LIN {X 0,Y 339.531,Z 433.374,A -85,B 0,C 180,E1 -14042.372,E2 -14042.372} C_VEL
LIN {X 0,Y 339.69,Z 432.812,A -85,B 0,C 180,E1 -14044.747,E2 -14044.747} C_VEL
LIN {X 0,Y 340.181,Z 431.007,A -85,B 0,C 180,E1 -14047.12,E2 -14047.12} C_VEL
LIN {X 0,Y 340.922,Z 427.934,A -85,B 0,C 180,E1 -14049.492,E2 -14049.492} C_VEL
LIN {X 0,Y 341.879,Z 423.539,A -85,B 0,C 180,E1 -14051.863,E2 -14051.863} C_VEL
LIN {X 0,Y 343.294,Z 417.733,A -85,B 0,C 180,E1 -14054.221,E2 -14054.221} C_VEL
LIN {X 0,Y 344.568,Z 412.354,A -85,B 0,C 180,E1 -14055.983,E2 -14055.983} C_VEL
LIN {X 0,Y 346.771,Z 403.681,A -85,B 0,C 180,E1 -14058.308,E2 -14058.308} C_VEL
LIN {X 0,Y 348.941,Z 394.494,A -85,B 0,C 180,E1 -14060.33,E2 -14060.33} C_VEL
LIN {X 0,Y 351.488,Z 383.498,A -85,B 0,C 180,E1 -14062.327,E2 -14062.327} C_VEL
LIN {X 0,Y 354.287,Z 371.267,A -85,B 0,C 180,E1 -14064.146,E2 -14064.146} C_VEL
LIN {X 0,Y 356.805,Z 358.929,A -85,B 0,C 180,E1 -14065.679,E2 -14065.679} C_VEL
LIN {X 0,Y 359.387,Z 345.597,A -85,B 0,C 180,E1 -14067.043,E2 -14067.043} C_VEL
LIN {X 0,Y 361.83,Z 331.122,A -85,B 0,C 180,E1 -14068.258,E2 -14068.258} C_VEL
LIN {X 0,Y 364.103,Z 316.147,A -85,B 0,C 180,E1 -14069.253,E2 -14069.253} C_VEL
LIN {X 0,Y 366.036,Z 300.525,A -85,B 0,C 180,E1 -14070.067,E2 -14070.067} C_VEL
LIN {X 0,Y 367.961,Z 282.022,A -85,B 0,C 180,E1 -14070.767,E2 -14070.767} C_VEL
LIN {X 0,Y 375.63,Z 216.607,A -85,B 0,C 180,E1 -14073.03,E2 -14073.03} C_VEL
LIN {X 0,Y 379.653,Z 185.862,A -85,B 0,C 180,E1 -14074.119,E2 -14074.119} C_VEL
LIN {X 0,Y 376.328,Z 179.523,A -85,B 0,C 180,E1 -14075.526,E2 -14075.526} C_VEL
LIN {X 0,Y 373.796,Z 175.547,A -85,B 0,C 180,E1 -14076.722,E2 -14076.722} C_VEL
LIN {X 0,Y 371.547,Z 172.279,A -85,B 0,C 180,E1 -14077.969,E2 -14077.969} C_VEL
LIN {X 0,Y 369.521,Z 169.583,A -85,B 0,C 180,E1 -14079.332,E2 -14079.332} C_VEL
LIN {X 0,Y 367.108,Z 166.762,A -85,B 0,C 180,E1 -14081.701,E2 -14081.701} C_VEL
LIN {X 0,Y 365.993,Z 166.623,A -85,B 0,C 180,E1 -14083.732,E2 -14083.732} C_VEL
LIN {X 0,Y 365.943,Z 167.567,A -85,B 0,C 180,E1 -14085.646,E2 -14085.646} C_VEL
LIN {X 0,Y 366.76,Z 169.742,A -85,B 0,C 180,E1 -14087.516,E2 -14087.516} C_VEL
LIN {X 0,Y 368.364,Z 172.942,A -85,B 0,C 180,E1 -14089.299,E2 -14089.299} C_VEL
LIN {X 0,Y 371.418,Z 179.732,A -85,B 0,C 180,E1 -14091.59,E2 -14091.59} C_VEL
LIN {X 0,Y 374.03,Z 186.01,A -85,B 0,C 180,E1 -14093.104,E2 -14093.104} C_VEL
LIN {X 0,Y 376.608,Z 193.132,A -85,B 0,C 180,E1 -14094.421,E2 -14094.421} C_VEL
LIN {X 0,Y 377.224,Z 207.224,A -85,B 0,C 180,E1 -14095.553,E2 -14095.553} C_VEL
LIN {X 0,Y 377.182,Z 212.766,A -85,B 0,C 180,E1 -14095.905,E2 -14095.905} C_VEL
LIN {X 0,Y 368.41,Z 287.792,A -85,B 0,C 180,E1 -14098.479,E2 -14098.479} C_VEL
LIN {X 0,Y 364.577,Z 324.529,A -85,B 0,C 180,E1 -14099.76,E2 -14099.76} C_VEL
LIN {X 0,Y 362.084,Z 341.748,A -85,B 0,C 180,E1 -14100.573,E2 -14100.573} C_VEL
LIN {X 0,Y 359.351,Z 357.417,A -85,B 0,C 180,E1 -14101.529,E2 -14101.529} C_VEL
LIN {X 0,Y 356.653,Z 371.828,A -85,B 0,C 180,E1 -14102.646,E2 -14102.646} C_VEL
LIN {X 0,Y 353.636,Z 386.742,A -85,B 0,C 180,E1 -14104.073,E2 -14104.073} C_VEL
LIN {X 0,Y 350.88,Z 399.866,A -85,B 0,C 180,E1 -14105.6,E2 -14105.6} C_VEL
LIN {X 0,Y 348.084,Z 412.984,A -85,B 0,C 180,E1 -14107.442,E2 -14107.442} C_VEL
LIN {X 0,Y 345.654,Z 424.786,A -85,B 0,C 180,E1 -14109.445,E2 -14109.445} C_VEL
LIN {X 0,Y 343.653,Z 435.782,A -85,B 0,C 180,E1 -14111.519,E2 -14111.519} C_VEL
LIN {X 0,Y 342.125,Z 444.941,A -85,B 0,C 180,E1 -14113.593,E2 -14113.593} C_VEL
LIN {X 0,Y 340.95,Z 452.532,A -85,B 0,C 180,E1 -14115.679,E2 -14115.679} C_VEL
LIN {X 0,Y 340.039,Z 459.612,A -85,B 0,C 180,E1 -14118.072,E2 -14118.072} C_VEL
LIN {X 0,Y 339.417,Z 465.159,A -85,B 0,C 180,E1 -14120.465,E2 -14120.465} C_VEL
LIN {X 0,Y 339.169,Z 469.321,A -85,B 0,C 180,E1 -14122.858,E2 -14122.858} C_VEL
LIN {X 0,Y 339.05,Z 472.204,A -85,B 0,C 180,E1 -14125.244,E2 -14125.244} C_VEL
LIN {X 0,Y 339.04,Z 473.874,A -85,B 0,C 180,E1 -14127.624,E2 -14127.624} C_VEL
LIN {X 0,Y 339.07,Z 474.355,A -85,B 0,C 180,E1 -14130,E2 -14130} C_VEL
LIN {X 0,Y 339.041,Z 473.645,A -85,B 0,C 180,E1 -14132.376,E2 -14132.376} C_VEL
LIN {X 0,Y 339.064,Z 471.711,A -85,B 0,C 180,E1 -14134.756,E2 -14134.756} C_VEL
LIN {X 0,Y 339.22,Z 468.501,A -85,B 0,C 180,E1 -14137.141,E2 -14137.141} C_VEL
LIN {X 0,Y 339.362,Z 463.965,A -85,B 0,C 180,E1 -14139.537,E2 -14139.537} C_VEL
LIN {X 0,Y 339.951,Z 458.003,A -85,B 0,C 180,E1 -14141.931,E2 -14141.931} C_VEL
LIN {X 0,Y 340.726,Z 450.427,A -85,B 0,C 180,E1 -14144.331,E2 -14144.331} C_VEL
LIN {X 0,Y 341.897,Z 442.263,A -85,B 0,C 180,E1 -14146.418,E2 -14146.418} C_VEL
LIN {X 0,Y 344.5,Z 427.37,A -85,B 0,C 180,E1 -14149.67,E2 -14149.67} C_VEL
LIN {X 0,Y 346.677,Z 416.152,A -85,B 0,C 180,E1 -14151.714,E2 -14151.714} C_VEL
LIN {X 0,Y 349.347,Z 403.732,A -85,B 0,C 180,E1 -14153.568,E2 -14153.568} C_VEL
LIN {X 0,Y 352.146,Z 390.155,A -85,B 0,C 180,E1 -14155.252,E2 -14155.252} C_VEL
LIN {X 0,Y 355.058,Z 375.843,A -85,B 0,C 180,E1 -14156.695,E2 -14156.695} C_VEL
LIN {X 0,Y 357.887,Z 360.455,A -85,B 0,C 180,E1 -14157.972,E2 -14157.972} C_VEL
LIN {X 0,Y 360.631,Z 344.612,A -85,B 0,C 180,E1 -14158.997,E2 -14158.997} C_VEL
LIN {X 0,Y 363.283,Z 326.693,A -85,B 0,C 180,E1 -14159.878,E2 -14159.878} C_VEL
LIN {X 0,Y 365.647,Z 304.905,A -85,B 0,C 180,E1 -14160.66,E2 -14160.66} C_VEL
LIN {X 0,Y 373.572,Z 232.695,A -85,B 0,C 180,E1 -14163.138,E2 -14163.138} C_VEL
LIN {X 0,Y 376.754,Z 206.525,A -85,B 0,C 180,E1 -14164.063,E2 -14164.063} C_VEL
LIN {X 0,Y 377.117,Z 189.528,A -85,B 0,C 180,E1 -14165.126,E2 -14165.126} C_VEL
LIN {X 0,Y 377.037,Z 185.508,A -85,B 0,C 180,E1 -14165.437,E2 -14165.437} C_VEL
LIN {X 0,Y 374.782,Z 174.187,A -85,B 0,C 180,E1 -14167.011,E2 -14167.011} C_VEL
LIN {X 0,Y 372.206,Z 169.945,A -85,B 0,C 180,E1 -14168.343,E2 -14168.343} C_VEL
LIN {X 0,Y 370.361,Z 166.78,A -85,B 0,C 180,E1 -14169.51,E2 -14169.51} C_VEL
LIN {X 0,Y 367.673,Z 162.482,A -85,B 0,C 180,E1 -14171.8,E2 -14171.8} C_VEL
LIN {X 0,Y 366.032,Z 160.666,A -85,B 0,C 180,E1 -14174.345,E2 -14174.345} C_VEL
LIN {X 0,Y 365.952,Z 160.508,A -85,B 0,C 180,E1 -14176.262,E2 -14176.262} C_VEL
LIN {X 0,Y 366.717,Z 161.339,A -85,B 0,C 180,E1 -14178.083,E2 -14178.083} C_VEL
LIN {X 0,Y 368.403,Z 163.16,A -85,B 0,C 180,E1 -14179.91,E2 -14179.91} C_VEL
LIN {X 0,Y 370.56,Z 166.521,A -85,B 0,C 180,E1 -14181.597,E2 -14181.597} C_VEL
LIN {X 0,Y 373.531,Z 171.452,A -85,B 0,C 180,E1 -14183.332,E2 -14183.332} C_VEL
LIN {X 0,Y 375.997,Z 175.941,A -85,B 0,C 180,E1 -14184.535,E2 -14184.535} C_VEL
LIN {X 0,Y 379.423,Z 182.777,A -85,B 0,C 180,E1 -14185.992,E2 -14185.992} C_VEL
LIN {X 0,Y 369.991,Z 258.966,A -85,B 0,C 180,E1 -14188.629,E2 -14188.629} C_VEL
LIN {X 0,Y 366.125,Z 295.865,A -85,B 0,C 180,E1 -14189.909,E2 -14189.909} C_VEL
LIN {X 0,Y 364.358,Z 311.193,A -85,B 0,C 180,E1 -14190.642,E2 -14190.642} C_VEL
LIN {X 0,Y 362.129,Z 326.807,A -85,B 0,C 180,E1 -14191.61,E2 -14191.61} C_VEL
LIN {X 0,Y 359.897,Z 340.486,A -85,B 0,C 180,E1 -14192.684,E2 -14192.684} C_VEL
LIN {X 0,Y 357.363,Z 354.596,A -85,B 0,C 180,E1 -14194.051,E2 -14194.051} C_VEL
LIN {X 0,Y 354.988,Z 366.509,A -85,B 0,C 180,E1 -14195.433,E2 -14195.433} C_VEL
LIN {X 0,Y 352.176,Z 379.037,A -85,B 0,C 180,E1 -14197.171,E2 -14197.171} C_VEL
LIN {X 0,Y 349.605,Z 390.384,A -85,B 0,C 180,E1 -14199.095,E2 -14199.095} C_VEL
LIN {X 0,Y 347.647,Z 398.906,A -85,B 0,C 180,E1 -14200.822,E2 -14200.822} C_VEL
LIN {X 0,Y 345.627,Z 407.42,A -85,B 0,C 180,E1 -14202.882,E2 -14202.882} C_VEL
LIN {X 0,Y 344.03,Z 413.434,A -85,B 0,C 180,E1 -14204.6,E2 -14204.6} C_VEL
LIN {X 0,Y 342.6,Z 420.079,A -85,B 0,C 180,E1 -14206.959,E2 -14206.959} C_VEL
LIN {X 0,Y 341.42,Z 425.246,A -85,B 0,C 180,E1 -14209.324,E2 -14209.324} C_VEL
LIN {X 0,Y 340.504,Z 429.044,A -85,B 0,C 180,E1 -14211.693,E2 -14211.693} C_VEL
LIN {X 0,Y 339.786,Z 431.564,A -85,B 0,C 180,E1 -14214.064,E2 -14214.064} C_VEL
LIN {X 0,Y 339.631,Z 432.805,A -85,B 0,C 180,E1 -14216.441,E2 -14216.441} C_VEL
LIN {X 0,Y 339.363,Z 432.834,A -85,B 0,C 180,E1 -14218.814,E2 -14218.814} C_VEL
LIN {X 0,Y 339.27,Z 431.606,A -85,B 0,C 180,E1 -14221.187,E2 -14221.187} C_VEL
LIN {X 0,Y 339.294,Z 429.111,A -85,B 0,C 180,E1 -14223.563,E2 -14223.563} C_VEL
LIN {X 0,Y 339.449,Z 425.282,A -85,B 0,C 180,E1 -14225.942,E2 -14225.942} C_VEL
LIN {X 0,Y 339.686,Z 421.495,A -85,B 0,C 180,E1 -14227.729,E2 -14227.729} C_VEL
LIN {X 0,Y 340.078,Z 415.107,A -85,B 0,C 180,E1 -14230.117,E2 -14230.117} C_VEL
LIN {X 0,Y 340.702,Z 408.102,A -85,B 0,C 180,E1 -14232.207,E2 -14232.207} C_VEL
LIN {X 0,Y 341.404,Z 399.606,A -85,B 0,C 180,E1 -14234.302,E2 -14234.302} C_VEL
LIN {X 0,Y 342.454,Z 389.382,A -85,B 0,C 180,E1 -14236.391,E2 -14236.391} C_VEL
LIN {X 0,Y 343.567,Z 378.89,A -85,B 0,C 180,E1 -14238.177,E2 -14238.177} C_VEL
LIN {X 0,Y 344.895,Z 366.418,A -85,B 0,C 180,E1 -14239.958,E2 -14239.958} C_VEL
LIN {X 0,Y 346.164,Z 353.994,A -85,B 0,C 180,E1 -14241.435,E2 -14241.435} C_VEL
LIN {X 0,Y 347.407,Z 340.598,A -85,B 0,C 180,E1 -14242.762,E2 -14242.762} C_VEL
LIN {X 0,Y 348.684,Z 326.049,A -85,B 0,C 180,E1 -14243.931,E2 -14243.931} C_VEL
LIN {X 0,Y 349.755,Z 311.213,A -85,B 0,C 180,E1 -14244.88,E2 -14244.88} C_VEL
LIN {X 0,Y 350.628,Z 295.257,A -85,B 0,C 180,E1 -14245.657,E2 -14245.657} C_VEL
LIN {X 0,Y 351.365,Z 278.358,A -85,B 0,C 180,E1 -14246.227,E2 -14246.227} C_VEL
LIN {X 0,Y 356.1,Z 165.117,A -85,B 0,C 180,E1 -14249.306,E2 -14249.306} C_VEL
LIN {X 0,Y 343.866,Z 136.506,A -85,B 0,C 180,E1 -14251.007,E2 -14251.007} C_VEL
LIN {X 0,Y 340.762,Z 128.926,A -85,B 0,C 180,E1 -14251.469,E2 -14251.469} C_VEL
LIN {X 0,Y 340.717,Z 128.671,A -85,B 0,C 180,E1 -14251.5,E2 -14251.5} C_VEL
LIN {X 0,Y 340.719,Z 128.67,A -85,B 0,C 180,E1 -14255.279,E2 -14255.279} C_VEL
LIN {X 0,Y 340.695,Z 128.67,A -85,B 0,C 180,E1 -14258.383,E2 -14258.383} C_VEL
LIN {X 0,Y 340.695,Z 128.671,A -85,B 0,C 180,E1 -14262.045,E2 -14262.045} C_VEL
LIN {X 0,Y 340.651,Z 128.647,A -85,B 0,C 180,E1 -14266.228,E2 -14266.228} C_VEL
LIN {X 0,Y 340.671,Z 128.663,A -85,B 0,C 180,E1 -14268.688,E2 -14268.688} C_VEL
LIN {X 0,Y 340.721,Z 128.664,A -85,B 0,C 180,E1 -14271.771,E2 -14271.771} C_VEL
LIN {X 0,Y 340.724,Z 128.654,A -85,B 0,C 180,E1 -14275.596,E2 -14275.596} C_VEL
LIN {X 0,Y 340.696,Z 128.665,A -85,B 0,C 180,E1 -14278.955,E2 -14278.955} C_VEL
LIN {X 0,Y 340.72,Z 128.671,A -85,B 0,C 180,E1 -14283.013,E2 -14283.013} C_VEL
LIN {X 0,Y 340.707,Z 128.662,A -85,B 0,C 180,E1 -14286.926,E2 -14286.926} C_VEL
LIN {X 0,Y 340.711,Z 128.661,A -85,B 0,C 180,E1 -14290.729,E2 -14290.729} C_VEL
LIN {X 0,Y 340.796,Z 128.653,A -85,B 0,C 180,E1 -14294.449,E2 -14294.449} C_VEL
LIN {X 0,Y 340.851,Z 128.653,A -85,B 0,C 180,E1 -14298.101,E2 -14298.101} C_VEL
LIN {X 0,Y 340.9,Z 128.65,A -85,B 0,C 180,E1 -14300.666,E2 -14300.666} C_VEL
LIN {X 0,Y 344.768,Z 141.178,A -85,B 0,C 180,E1 -14303.295,E2 -14303.295} C_VEL
LIN {X 0,Y 345.612,Z 144.445,A -85,B 0,C 180,E1 -14303.958,E2 -14303.958} C_VEL
LIN {X 0,Y 354.099,Z 162.889,A -85,B 0,C 180,E1 -14305.218,E2 -14305.218} C_VEL
LIN {X 0,Y 358.782,Z 174.501,A -85,B 0,C 180,E1 -14305.916,E2 -14305.916} C_VEL
LIN {X 0,Y 360.448,Z 183.181,A -85,B 0,C 180,E1 -14306.265,E2 -14306.265} C_VEL
LIN {X 0,Y 356.697,Z 311.468,A -85,B 0,C 180,E1 -14308.906,E2 -14308.906} C_VEL
LIN {X 0,Y 355.794,Z 326.954,A -85,B 0,C 180,E1 -14309.434,E2 -14309.434} C_VEL
LIN {X 0,Y 354.704,Z 341.289,A -85,B 0,C 180,E1 -14310.142,E2 -14310.142} C_VEL
LIN {X 0,Y 353.381,Z 354.6,A -85,B 0,C 180,E1 -14310.997,E2 -14310.997} C_VEL
LIN {X 0,Y 351.781,Z 368.118,A -85,B 0,C 180,E1 -14312.095,E2 -14312.095} C_VEL
LIN {X 0,Y 349.949,Z 381.572,A -85,B 0,C 180,E1 -14313.454,E2 -14313.454} C_VEL
LIN {X 0,Y 348.192,Z 393.498,A -85,B 0,C 180,E1 -14314.921,E2 -14314.921} C_VEL
LIN {X 0,Y 346.611,Z 403.302,A -85,B 0,C 180,E1 -14316.356,E2 -14316.356} C_VEL
LIN {X 0,Y 345.295,Z 407.535,A -85,B 0,C 180,E1 -14317.004,E2 -14317.004} C_VEL
LIN {X 0,Y 341.431,Z 414.164,A -85,B 0,C 180,E1 -14318.055,E2 -14318.055} C_VEL
LIN {X 0,Y 337.583,Z 420.443,A -85,B 0,C 180,E1 -14319.187,E2 -14319.187} C_VEL
LIN {X 0,Y 336.307,Z 423.969,A -85,B 0,C 180,E1 -14319.955,E2 -14319.955} C_VEL
LIN {X 0,Y 334.95,Z 432.269,A -85,B 0,C 180,E1 -14322.112,E2 -14322.112} C_VEL
LIN {X 0,Y 333.839,Z 439.575,A -85,B 0,C 180,E1 -14324.441,E2 -14324.441} C_VEL
LIN {X 0,Y 333.057,Z 444.901,A -85,B 0,C 180,E1 -14326.551,E2 -14326.551} C_VEL
LIN {X 0,Y 332.438,Z 449.981,A -85,B 0,C 180,E1 -14329.128,E2 -14329.128} C_VEL
LIN {X 0,Y 331.985,Z 453.172,A -85,B 0,C 180,E1 -14331.334,E2 -14331.334} C_VEL
LIN {X 0,Y 331.749,Z 455.509,A -85,B 0,C 180,E1 -14333.735,E2 -14333.735} C_VEL
LIN {X 0,Y 331.656,Z 456.752,A -85,B 0,C 180,E1 -14336.424,E2 -14336.424} C_VEL
LIN {X 0,Y 331.736,Z 456.573,A -85,B 0,C 180,E1 -14339.161,E2 -14339.161} C_VEL
LIN {X 0,Y 331.806,Z 455.925,A -85,B 0,C 180,E1 -14340.554,E2 -14340.554} C_VEL
LIN {X 0,Y 331.95,Z 454.74,A -85,B 0,C 180,E1 -14342.126,E2 -14342.126} C_VEL
LIN {X 0,Y 332.494,Z 451.586,A -85,B 0,C 180,E1 -14344.799,E2 -14344.799} C_VEL
LIN {X 0,Y 333.037,Z 447.607,A -85,B 0,C 180,E1 -14347.135,E2 -14347.135} C_VEL
LIN {X 0,Y 333.807,Z 443.151,A -85,B 0,C 180,E1 -14349.17,E2 -14349.17} C_VEL
LIN {X 0,Y 334.912,Z 436.919,A -85,B 0,C 180,E1 -14351.451,E2 -14351.451} C_VEL
LIN {X 0,Y 336.282,Z 429.661,A -85,B 0,C 180,E1 -14353.604,E2 -14353.604} C_VEL
LIN {X 0,Y 338.119,Z 420.561,A -85,B 0,C 180,E1 -14355.816,E2 -14355.816} C_VEL
LIN {X 0,Y 339.994,Z 411.142,A -85,B 0,C 180,E1 -14357.704,E2 -14357.704} C_VEL
LIN {X 0,Y 342.016,Z 400.485,A -85,B 0,C 180,E1 -14359.491,E2 -14359.491} C_VEL
LIN {X 0,Y 344.214,Z 388.76,A -85,B 0,C 180,E1 -14361.116,E2 -14361.116} C_VEL
LIN {X 0,Y 346.492,Z 375.099,A -85,B 0,C 180,E1 -14362.67,E2 -14362.67} C_VEL
LIN {X 0,Y 348.48,Z 361.74,A -85,B 0,C 180,E1 -14363.893,E2 -14363.893} C_VEL
LIN {X 0,Y 350.282,Z 346.956,A -85,B 0,C 180,E1 -14364.965,E2 -14364.965} C_VEL
LIN {X 0,Y 351.786,Z 331.9,A -85,B 0,C 180,E1 -14365.787,E2 -14365.787} C_VEL
LIN {X 0,Y 352.835,Z 317.283,A -85,B 0,C 180,E1 -14366.36,E2 -14366.36} C_VEL
LIN {X 0,Y 353.595,Z 298.521,A -85,B 0,C 180,E1 -14366.825,E2 -14366.825} C_VEL
LIN {X 0,Y 357.635,Z 180.373,A -85,B 0,C 180,E1 -14369.304,E2 -14369.304} C_VEL
LIN {X 0,Y 354.976,Z 174.067,A -85,B 0,C 180,E1 -14369.766,E2 -14369.766} C_VEL
LIN {X 0,Y 354.401,Z 173.922,A -85,B 0,C 180,E1 -14369.836,E2 -14369.836} C_VEL
LIN {X 0,Y 352.541,Z 176.084,A -85,B 0,C 180,E1 -14369.997,E2 -14369.997} C_VEL
LIN {X 0,Y 351.147,Z 176.208,A -85,B 0,C 180,E1 -14370.158,E2 -14370.158} C_VEL
LIN {X 0,Y 350.137,Z 175.013,A -85,B 0,C 180,E1 -14370.31,E2 -14370.31} C_VEL
LIN {X 0,Y 349.399,Z 171.848,A -85,B 0,C 180,E1 -14370.496,E2 -14370.496} C_VEL
LIN {X 0,Y 344.234,Z 289.337,A -85,B 0,C 180,E1 -14373.832,E2 -14373.832} C_VEL
LIN {X 0,Y 343.353,Z 305.603,A -85,B 0,C 180,E1 -14374.542,E2 -14374.542} C_VEL
LIN {X 0,Y 342.32,Z 320.697,A -85,B 0,C 180,E1 -14375.433,E2 -14375.433} C_VEL
LIN {X 0,Y 341.032,Z 336.391,A -85,B 0,C 180,E1 -14376.627,E2 -14376.627} C_VEL
LIN {X 0,Y 339.665,Z 350.616,A -85,B 0,C 180,E1 -14377.974,E2 -14377.974} C_VEL
LIN {X 0,Y 338.34,Z 363.696,A -85,B 0,C 180,E1 -14379.48,E2 -14379.48} C_VEL
LIN {X 0,Y 337.035,Z 375.747,A -85,B 0,C 180,E1 -14381.142,E2 -14381.142} C_VEL
LIN {X 0,Y 335.843,Z 386.83,A -85,B 0,C 180,E1 -14382.964,E2 -14382.964} C_VEL
LIN {X 0,Y 334.696,Z 397.2,A -85,B 0,C 180,E1 -14384.998,E2 -14384.998} C_VEL
LIN {X 0,Y 334.024,Z 405.411,A -85,B 0,C 180,E1 -14386.927,E2 -14386.927} C_VEL
LIN {X 0,Y 333.199,Z 413.019,A -85,B 0,C 180,E1 -14389.057,E2 -14389.057} C_VEL
LIN {X 0,Y 332.7,Z 420.057,A -85,B 0,C 180,E1 -14391.496,E2 -14391.496} C_VEL
LIN {X 0,Y 332.373,Z 425.501,A -85,B 0,C 180,E1 -14393.931,E2 -14393.931} C_VEL
LIN {X 0,Y 332.249,Z 429.507,A -85,B 0,C 180,E1 -14396.361,E2 -14396.361} C_VEL
LIN {X 0,Y 332.197,Z 432.193,A -85,B 0,C 180,E1 -14398.787,E2 -14398.787} C_VEL
LIN {X 0,Y 332.314,Z 433.61,A -85,B 0,C 180,E1 -14401.211,E2 -14401.211} C_VEL
LIN {X 0,Y 332.597,Z 433.782,A -85,B 0,C 180,E1 -14403.634,E2 -14403.634} C_VEL
LIN {X 0,Y 332.785,Z 432.739,A -85,B 0,C 180,E1 -14406.061,E2 -14406.061} C_VEL
LIN {X 0,Y 333.555,Z 430.397,A -85,B 0,C 180,E1 -14408.481,E2 -14408.481} C_VEL
LIN {X 0,Y 334.518,Z 426.792,A -85,B 0,C 180,E1 -14410.899,E2 -14410.899} C_VEL
LIN {X 0,Y 335.767,Z 421.865,A -85,B 0,C 180,E1 -14413.311,E2 -14413.311} C_VEL
LIN {X 0,Y 337.321,Z 415.514,A -85,B 0,C 180,E1 -14415.715,E2 -14415.715} C_VEL
LIN {X 0,Y 339.598,Z 407.5,A -85,B 0,C 180,E1 -14418.085,E2 -14418.085} C_VEL
LIN {X 0,Y 341.801,Z 398.991,A -85,B 0,C 180,E1 -14420.145,E2 -14420.145} C_VEL
LIN {X 0,Y 344.01,Z 390.384,A -85,B 0,C 180,E1 -14421.891,E2 -14421.891} C_VEL
LIN {X 0,Y 346.539,Z 380.333,A -85,B 0,C 180,E1 -14423.612,E2 -14423.612} C_VEL
LIN {X 0,Y 349.545,Z 367.455,A -85,B 0,C 180,E1 -14425.453,E2 -14425.453} C_VEL
LIN {X 0,Y 352.399,Z 354.435,A -85,B 0,C 180,E1 -14426.982,E2 -14426.982} C_VEL
LIN {X 0,Y 355.202,Z 340.288,A -85,B 0,C 180,E1 -14428.35,E2 -14428.35} C_VEL
LIN {X 0,Y 357.834,Z 325.147,A -85,B 0,C 180,E1 -14429.527,E2 -14429.527} C_VEL
LIN {X 0,Y 360.231,Z 309.373,A -85,B 0,C 180,E1 -14430.481,E2 -14430.481} C_VEL
LIN {X 0,Y 362.139,Z 293.588,A -85,B 0,C 180,E1 -14431.216,E2 -14431.216} C_VEL
LIN {X 0,Y 370.888,Z 223.056,A -85,B 0,C 180,E1 -14433.727,E2 -14433.727} C_VEL
LIN {X 0,Y 375.623,Z 189.779,A -85,B 0,C 180,E1 -14434.914,E2 -14434.914} C_VEL
LIN {X 0,Y 372.715,Z 184.281,A -85,B 0,C 180,E1 -14436.277,E2 -14436.277} C_VEL
LIN {X 0,Y 370.768,Z 181.122,A -85,B 0,C 180,E1 -14437.305,E2 -14437.305} C_VEL
LIN {X 0,Y 368.935,Z 178.392,A -85,B 0,C 180,E1 -14438.427,E2 -14438.427} C_VEL
LIN {X 0,Y 367.528,Z 176.346,A -85,B 0,C 180,E1 -14439.462,E2 -14439.462} C_VEL
LIN {X 0,Y 365.154,Z 173.57,A -85,B 0,C 180,E1 -14441.942,E2 -14441.942} C_VEL
LIN {X 0,Y 364.124,Z 173.703,A -85,B 0,C 180,E1 -14444.427,E2 -14444.427} C_VEL
LIN {X 0,Y 364.417,Z 175.29,A -85,B 0,C 180,E1 -14446.441,E2 -14446.441} C_VEL
LIN {X 0,Y 365.931,Z 178.684,A -85,B 0,C 180,E1 -14448.688,E2 -14448.688} C_VEL
LIN {X 0,Y 368.629,Z 185.213,A -85,B 0,C 180,E1 -14451.039,E2 -14451.039} C_VEL
LIN {X 0,Y 370.974,Z 191.486,A -85,B 0,C 180,E1 -14452.586,E2 -14452.586} C_VEL
LIN {X 0,Y 372.965,Z 197.371,A -85,B 0,C 180,E1 -14453.72,E2 -14453.72} C_VEL
LIN {X 0,Y 373.246,Z 210.584,A -85,B 0,C 180,E1 -14454.803,E2 -14454.803} C_VEL
LIN {X 0,Y 373.102,Z 214.773,A -85,B 0,C 180,E1 -14455.059,E2 -14455.059} C_VEL
LIN {X 0,Y 363.955,Z 287.115,A -85,B 0,C 180,E1 -14457.598,E2 -14457.598} C_VEL
LIN {X 0,Y 359.778,Z 323.576,A -85,B 0,C 180,E1 -14458.906,E2 -14458.906} C_VEL
LIN {X 0,Y 357.148,Z 340.609,A -85,B 0,C 180,E1 -14459.718,E2 -14459.718} C_VEL
LIN {X 0,Y 354.455,Z 355.202,A -85,B 0,C 180,E1 -14460.611,E2 -14460.611} C_VEL
LIN {X 0,Y 351.694,Z 369.012,A -85,B 0,C 180,E1 -14461.67,E2 -14461.67} C_VEL
LIN {X 0,Y 348.612,Z 383.461,A -85,B 0,C 180,E1 -14463.025,E2 -14463.025} C_VEL
LIN {X 0,Y 345.537,Z 396.919,A -85,B 0,C 180,E1 -14464.553,E2 -14464.553} C_VEL
LIN {X 0,Y 342.508,Z 410.357,A -85,B 0,C 180,E1 -14466.414,E2 -14466.414} C_VEL
LIN {X 0,Y 340.069,Z 420.922,A -85,B 0,C 180,E1 -14468.161,E2 -14468.161} C_VEL
LIN {X 0,Y 337.751,Z 431.458,A -85,B 0,C 180,E1 -14470.237,E2 -14470.237} C_VEL
LIN {X 0,Y 335.706,Z 442.451,A -85,B 0,C 180,E1 -14472.643,E2 -14472.643} C_VEL
LIN {X 0,Y 334.324,Z 450.434,A -85,B 0,C 180,E1 -14474.766,E2 -14474.766} C_VEL
LIN {X 0,Y 333.238,Z 457.89,A -85,B 0,C 180,E1 -14477.206,E2 -14477.206} C_VEL
LIN {X 0,Y 332.473,Z 463.786,A -85,B 0,C 180,E1 -14479.649,E2 -14479.649} C_VEL
LIN {X 0,Y 332.216,Z 467.283,A -85,B 0,C 180,E1 -14481.484,E2 -14481.484} C_VEL
LIN {X 0,Y 332.018,Z 471.102,A -85,B 0,C 180,E1 -14484.193,E2 -14484.193} C_VEL
LIN {X 0,Y 331.992,Z 473.027,A -85,B 0,C 180,E1 -14486.359,E2 -14486.359} C_VEL
LIN {X 0,Y 331.941,Z 474.08,A -85,B 0,C 180,E1 -14488.787,E2 -14488.787} C_VEL
LIN {X 0,Y 331.942,Z 473.947,A -85,B 0,C 180,E1 -14491.213,E2 -14491.213} C_VEL
LIN {X 0,Y 331.999,Z 472.62,A -85,B 0,C 180,E1 -14493.641,E2 -14493.641} C_VEL
LIN {X 0,Y 332.033,Z 470.034,A -85,B 0,C 180,E1 -14496.075,E2 -14496.075} C_VEL
LIN {X 0,Y 332.195,Z 466.148,A -85,B 0,C 180,E1 -14498.516,E2 -14498.516} C_VEL
LIN {X 0,Y 332.543,Z 460.887,A -85,B 0,C 180,E1 -14500.965,E2 -14500.965} C_VEL
LIN {X 0,Y 333.332,Z 454.119,A -85,B 0,C 180,E1 -14503.41,E2 -14503.41} C_VEL
LIN {X 0,Y 334.289,Z 446.76,A -85,B 0,C 180,E1 -14505.548,E2 -14505.548} C_VEL
LIN {X 0,Y 336.731,Z 433.47,A -85,B 0,C 180,E1 -14508.875,E2 -14508.875} C_VEL
LIN {X 0,Y 338.735,Z 423.704,A -85,B 0,C 180,E1 -14510.943,E2 -14510.943} C_VEL
LIN {X 0,Y 340.97,Z 413.547,A -85,B 0,C 180,E1 -14512.735,E2 -14512.735} C_VEL
LIN {X 0,Y 343.908,Z 400.888,A -85,B 0,C 180,E1 -14514.606,E2 -14514.606} C_VEL
LIN {X 0,Y 346.74,Z 388.206,A -85,B 0,C 180,E1 -14516.158,E2 -14516.158} C_VEL
LIN {X 0,Y 349.681,Z 374.7,A -85,B 0,C 180,E1 -14517.533,E2 -14517.533} C_VEL
LIN {X 0,Y 352.513,Z 360.213,A -85,B 0,C 180,E1 -14518.749,E2 -14518.749} C_VEL
LIN {X 0,Y 355.465,Z 344.586,A -85,B 0,C 180,E1 -14519.785,E2 -14519.785} C_VEL
LIN {X 0,Y 358.137,Z 327.899,A -85,B 0,C 180,E1 -14520.638,E2 -14520.638} C_VEL
LIN {X 0,Y 360.577,Z 308.25,A -85,B 0,C 180,E1 -14521.384,E2 -14521.384} C_VEL
LIN {X 0,Y 368.657,Z 239.15,A -85,B 0,C 180,E1 -14523.813,E2 -14523.813} C_VEL
LIN {X 0,Y 372.774,Z 207.982,A -85,B 0,C 180,E1 -14524.937,E2 -14524.937} C_VEL
LIN {X 0,Y 373.394,Z 191.654,A -85,B 0,C 180,E1 -14525.993,E2 -14525.993} C_VEL
LIN {X 0,Y 373.329,Z 188.885,A -85,B 0,C 180,E1 -14526.226,E2 -14526.226} C_VEL
LIN {X 0,Y 371.68,Z 179.651,A -85,B 0,C 180,E1 -14527.562,E2 -14527.562} C_VEL
LIN {X 0,Y 369.438,Z 175.772,A -85,B 0,C 180,E1 -14528.845,E2 -14528.845} C_VEL
LIN {X 0,Y 368.069,Z 173.302,A -85,B 0,C 180,E1 -14529.786,E2 -14529.786} C_VEL
LIN {X 0,Y 365.79,Z 169.302,A -85,B 0,C 180,E1 -14531.893,E2 -14531.893} C_VEL
LIN {X 0,Y 364.228,Z 167.504,A -85,B 0,C 180,E1 -14534.444,E2 -14534.444} C_VEL
LIN {X 0,Y 364.247,Z 167.416,A -85,B 0,C 180,E1 -14536.543,E2 -14536.543} C_VEL
LIN {X 0,Y 365.145,Z 168.486,A -85,B 0,C 180,E1 -14538.359,E2 -14538.359} C_VEL
LIN {X 0,Y 366.403,Z 169.869,A -85,B 0,C 180,E1 -14539.721,E2 -14539.721} C_VEL
LIN {X 0,Y 368.346,Z 173.103,A -85,B 0,C 180,E1 -14541.366,E2 -14541.366} C_VEL
LIN {X 0,Y 370.979,Z 177.752,A -85,B 0,C 180,E1 -14543.007,E2 -14543.007} C_VEL
LIN {X 0,Y 373.227,Z 182.091,A -85,B 0,C 180,E1 -14544.184,E2 -14544.184} C_VEL
LIN {X 0,Y 375.33,Z 186.552,A -85,B 0,C 180,E1 -14545.171,E2 -14545.171} C_VEL
LIN {X 0,Y 365.497,Z 260.26,A -85,B 0,C 180,E1 -14547.792,E2 -14547.792} C_VEL
LIN {X 0,Y 361.308,Z 297.057,A -85,B 0,C 180,E1 -14549.108,E2 -14549.108} C_VEL
LIN {X 0,Y 359.559,Z 310.857,A -85,B 0,C 180,E1 -14549.782,E2 -14549.782} C_VEL
LIN {X 0,Y 357.308,Z 325.755,A -85,B 0,C 180,E1 -14550.707,E2 -14550.707} C_VEL
LIN {X 0,Y 354.898,Z 339.586,A -85,B 0,C 180,E1 -14551.785,E2 -14551.785} C_VEL
LIN {X 0,Y 352.174,Z 353.869,A -85,B 0,C 180,E1 -14553.16,E2 -14553.16} C_VEL
LIN {X 0,Y 349.381,Z 366.948,A -85,B 0,C 180,E1 -14554.694,E2 -14554.694} C_VEL
LIN {X 0,Y 346.504,Z 378.984,A -85,B 0,C 180,E1 -14556.386,E2 -14556.386} C_VEL
LIN {X 0,Y 344.003,Z 389.196,A -85,B 0,C 180,E1 -14558.109,E2 -14558.109} C_VEL
LIN {X 0,Y 341.75,Z 397.939,A -85,B 0,C 180,E1 -14559.852,E2 -14559.852} C_VEL
LIN {X 0,Y 339.596,Z 406.543,A -85,B 0,C 180,E1 -14561.915,E2 -14561.915} C_VEL
LIN {X 0,Y 337.299,Z 414.7,A -85,B 0,C 180,E1 -14564.284,E2 -14564.284} C_VEL
LIN {X 0,Y 335.757,Z 421.152,A -85,B 0,C 180,E1 -14566.689,E2 -14566.689} C_VEL
LIN {X 0,Y 334.496,Z 426.168,A -85,B 0,C 180,E1 -14569.1,E2 -14569.1} C_VEL
LIN {X 0,Y 333.52,Z 429.834,A -85,B 0,C 180,E1 -14571.518,E2 -14571.518} C_VEL
LIN {X 0,Y 332.758,Z 432.221,A -85,B 0,C 180,E1 -14573.938,E2 -14573.938} C_VEL
LIN {X 0,Y 332.55,Z 433.333,A -85,B 0,C 180,E1 -14576.365,E2 -14576.365} C_VEL
LIN {X 0,Y 332.288,Z 433.227,A -85,B 0,C 180,E1 -14578.788,E2 -14578.788} C_VEL
LIN {X 0,Y 332.175,Z 431.872,A -85,B 0,C 180,E1 -14581.213,E2 -14581.213} C_VEL
LIN {X 0,Y 332.215,Z 429.243,A -85,B 0,C 180,E1 -14583.639,E2 -14583.639} C_VEL
LIN {X 0,Y 332.366,Z 425.277,A -85,B 0,C 180,E1 -14586.069,E2 -14586.069} C_VEL
LIN {X 0,Y 332.61,Z 421.409,A -85,B 0,C 180,E1 -14587.895,E2 -14587.895} C_VEL
LIN {X 0,Y 333.033,Z 414.836,A -85,B 0,C 180,E1 -14590.334,E2 -14590.334} C_VEL
LIN {X 0,Y 333.824,Z 406.517,A -85,B 0,C 180,E1 -14592.772,E2 -14592.772} C_VEL
LIN {X 0,Y 334.534,Z 397.656,A -85,B 0,C 180,E1 -14594.898,E2 -14594.898} C_VEL
LIN {X 0,Y 335.527,Z 388.514,A -85,B 0,C 180,E1 -14596.739,E2 -14596.739} C_VEL
LIN {X 0,Y 336.818,Z 376.792,A -85,B 0,C 180,E1 -14598.713,E2 -14598.713} C_VEL
LIN {X 0,Y 338.092,Z 364.973,A -85,B 0,C 180,E1 -14600.377,E2 -14600.377} C_VEL
LIN {X 0,Y 339.458,Z 352.212,A -85,B 0,C 180,E1 -14601.881,E2 -14601.881} C_VEL
LIN {X 0,Y 340.738,Z 338.368,A -85,B 0,C 180,E1 -14603.233,E2 -14603.233} C_VEL
LIN {X 0,Y 342.037,Z 323.232,A -85,B 0,C 180,E1 -14604.427,E2 -14604.427} C_VEL
LIN {X 0,Y 343.118,Z 307.555,A -85,B 0,C 180,E1 -14605.396,E2 -14605.396} C_VEL
LIN {X 0,Y 344.022,Z 291.666,A -85,B 0,C 180,E1 -14606.125,E2 -14606.125} C_VEL
LIN {X 0,Y 344.894,Z 271.105,A -85,B 0,C 180,E1 -14606.758,E2 -14606.758} C_VEL
LIN {X 0,Y 349.36,Z 166.325,A -85,B 0,C 180,E1 -14609.7,E2 -14609.7} C_VEL
LIN {X 0,Y 333.698,Z 129.829,A -85,B 0,C 180,E1 -14611.952,E2 -14611.952} C_VEL
LIN {X 0,Y 333.674,Z 129.548,A -85,B 0,C 180,E1 -14612.041,E2 -14612.041} C_VEL
LIN {X 0,Y 333.687,Z 129.544,A -85,B 0,C 180,E1 -14614.774,E2 -14614.774} C_VEL
LIN {X 0,Y 333.645,Z 129.551,A -85,B 0,C 180,E1 -14617.653,E2 -14617.653} C_VEL
LIN {X 0,Y 333.605,Z 129.554,A -85,B 0,C 180,E1 -14620.774,E2 -14620.774} C_VEL
LIN {X 0,Y 333.592,Z 129.548,A -85,B 0,C 180,E1 -14624.25,E2 -14624.25} C_VEL
LIN {X 0,Y 333.638,Z 129.525,A -85,B 0,C 180,E1 -14627.618,E2 -14627.618} C_VEL
LIN {X 0,Y 333.636,Z 129.551,A -85,B 0,C 180,E1 -14631.206,E2 -14631.206} C_VEL
LIN {X 0,Y 333.676,Z 129.522,A -85,B 0,C 180,E1 -14633.861,E2 -14633.861} C_VEL
LIN {X 0,Y 333.646,Z 129.55,A -85,B 0,C 180,E1 -14637.413,E2 -14637.413} C_VEL
LIN {X 0,Y 333.655,Z 129.532,A -85,B 0,C 180,E1 -14641.023,E2 -14641.023} C_VEL
LIN {X 0,Y 333.665,Z 129.535,A -85,B 0,C 180,E1 -14645.086,E2 -14645.086} C_VEL
LIN {X 0,Y 333.658,Z 129.544,A -85,B 0,C 180,E1 -14649.018,E2 -14649.018} C_VEL
LIN {X 0,Y 333.716,Z 129.541,A -85,B 0,C 180,E1 -14651.585,E2 -14651.585} C_VEL
LIN {X 0,Y 333.777,Z 129.536,A -85,B 0,C 180,E1 -14655.6,E2 -14655.6} C_VEL
LIN {X 0,Y 333.819,Z 129.525,A -85,B 0,C 180,E1 -14659.078,E2 -14659.078} C_VEL
LIN {X 0,Y 333.82,Z 129.605,A -85,B 0,C 180,E1 -14660.036,E2 -14660.036} C_VEL
LIN {X 0,Y 338.333,Z 143.961,A -85,B 0,C 180,E1 -14663.11,E2 -14663.11} C_VEL
LIN {X 0,Y 338.717,Z 145.145,A -85,B 0,C 180,E1 -14663.284,E2 -14663.284} C_VEL
LIN {X 0,Y 348.433,Z 166.103,A -85,B 0,C 180,E1 -14664.766,E2 -14664.766} C_VEL
LIN {X 0,Y 352.899,Z 177.405,A -85,B 0,C 180,E1 -14665.454,E2 -14665.454} C_VEL
LIN {X 0,Y 354.215,Z 184.577,A -85,B 0,C 180,E1 -14665.744,E2 -14665.744} C_VEL
LIN {X 0,Y 350.313,Z 312.251,A -85,B 0,C 180,E1 -14668.419,E2 -14668.419} C_VEL
LIN {X 0,Y 349.368,Z 327.564,A -85,B 0,C 180,E1 -14668.955,E2 -14668.955} C_VEL
LIN {X 0,Y 348.182,Z 342.4,A -85,B 0,C 180,E1 -14669.711,E2 -14669.711} C_VEL
LIN {X 0,Y 346.578,Z 357.409,A -85,B 0,C 180,E1 -14670.726,E2 -14670.726} C_VEL
LIN {X 0,Y 344.946,Z 370.834,A -85,B 0,C 180,E1 -14671.888,E2 -14671.888} C_VEL
LIN {X 0,Y 343.075,Z 383.51,A -85,B 0,C 180,E1 -14673.229,E2 -14673.229} C_VEL
LIN {X 0,Y 341.09,Z 396.213,A -85,B 0,C 180,E1 -14674.876,E2 -14674.876} C_VEL
LIN {X 0,Y 339.138,Z 407.667,A -85,B 0,C 180,E1 -14676.675,E2 -14676.675} C_VEL
LIN {X 0,Y 337.329,Z 418.238,A -85,B 0,C 180,E1 -14678.688,E2 -14678.688} C_VEL
LIN {X 0,Y 336.307,Z 423.969,A -85,B 0,C 180,E1 -14679.955,E2 -14679.955} C_VEL
LIN {X 0,Y 335.071,Z 427.407,A -85,B 0,C 180,E1 -14680.748,E2 -14680.748} C_VEL
LIN {X 0,Y 331.405,Z 432.659,A -85,B 0,C 180,E1 -14682.051,E2 -14682.051} C_VEL
LIN {X 0,Y 327.834,Z 437.451,A -85,B 0,C 180,E1 -14683.432,E2 -14683.432} C_VEL
LIN {X 0,Y 326.764,Z 440.1,A -85,B 0,C 180,E1 -14684.337,E2 -14684.337} C_VEL
LIN {X 0,Y 325.859,Z 446.334,A -85,B 0,C 180,E1 -14686.928,E2 -14686.928} C_VEL
LIN {X 0,Y 325.241,Z 451.099,A -85,B 0,C 180,E1 -14689.569,E2 -14689.569} C_VEL
LIN {X 0,Y 324.858,Z 453.735,A -85,B 0,C 180,E1 -14691.579,E2 -14691.579} C_VEL
LIN {X 0,Y 324.64,Z 456.068,A -85,B 0,C 180,E1 -14694.288,E2 -14694.288} C_VEL
LIN {X 0,Y 324.561,Z 457.021,A -85,B 0,C 180,E1 -14697.048,E2 -14697.048} C_VEL
LIN {X 0,Y 324.611,Z 456.964,A -85,B 0,C 180,E1 -14698.445,E2 -14698.445} C_VEL
LIN {X 0,Y 324.679,Z 456.48,A -85,B 0,C 180,E1 -14700.02,E2 -14700.02} C_VEL
LIN {X 0,Y 324.943,Z 454.534,A -85,B 0,C 180,E1 -14702.732,E2 -14702.732} C_VEL
LIN {X 0,Y 325.432,Z 451.996,A -85,B 0,C 180,E1 -14704.85,E2 -14704.85} C_VEL
LIN {X 0,Y 325.953,Z 448.3,A -85,B 0,C 180,E1 -14707.137,E2 -14707.137} C_VEL
LIN {X 0,Y 326.927,Z 442.928,A -85,B 0,C 180,E1 -14709.643,E2 -14709.643} C_VEL
LIN {X 0,Y 328.135,Z 436.46,A -85,B 0,C 180,E1 -14712.014,E2 -14712.014} C_VEL
LIN {X 0,Y 329.752,Z 428.661,A -85,B 0,C 180,E1 -14714.316,E2 -14714.316} C_VEL
LIN {X 0,Y 331.727,Z 419.495,A -85,B 0,C 180,E1 -14716.521,E2 -14716.521} C_VEL
LIN {X 0,Y 333.846,Z 409.06,A -85,B 0,C 180,E1 -14718.587,E2 -14718.587} C_VEL
LIN {X 0,Y 335.93,Z 398.74,A -85,B 0,C 180,E1 -14720.288,E2 -14720.288} C_VEL
LIN {X 0,Y 338.26,Z 386.362,A -85,B 0,C 180,E1 -14721.976,E2 -14721.976} C_VEL
LIN {X 0,Y 340.514,Z 373.383,A -85,B 0,C 180,E1 -14723.418,E2 -14723.418} C_VEL
LIN {X 0,Y 342.566,Z 359.821,A -85,B 0,C 180,E1 -14724.637,E2 -14724.637} C_VEL
LIN {X 0,Y 344.305,Z 345.939,A -85,B 0,C 180,E1 -14725.63,E2 -14725.63} C_VEL
LIN {X 0,Y 345.812,Z 330.518,A -85,B 0,C 180,E1 -14726.465,E2 -14726.465} C_VEL
LIN {X 0,Y 346.958,Z 315.119,A -85,B 0,C 180,E1 -14727.04,E2 -14727.04} C_VEL
LIN {X 0,Y 347.985,Z 287.959,A -85,B 0,C 180,E1 -14727.669,E2 -14727.669} C_VEL
LIN {X 0,Y 351.646,Z 186.622,A -85,B 0,C 180,E1 -14729.83,E2 -14729.83} C_VEL
LIN {X 0,Y 348.279,Z 195.922,A -85,B 0,C 180,E1 -14729.986,E2 -14729.986} C_VEL
LIN {X 0,Y 345.833,Z 200.401,A -85,B 0,C 180,E1 -14730.161,E2 -14730.161} C_VEL
LIN {X 0,Y 344.175,Z 201.783,A -85,B 0,C 180,E1 -14730.325,E2 -14730.325} C_VEL
LIN {X 0,Y 343.096,Z 201.658,A -85,B 0,C 180,E1 -14730.46,E2 -14730.46} C_VEL
LIN {X 0,Y 342.086,Z 200.124,A -85,B 0,C 180,E1 -14730.626,E2 -14730.626} C_VEL
LIN {X 0,Y 341.49,Z 197.114,A -85,B 0,C 180,E1 -14730.781,E2 -14730.781} C_VEL
LIN {X 0,Y 337.367,Z 290.173,A -85,B 0,C 180,E1 -14733.532,E2 -14733.532} C_VEL
LIN {X 0,Y 336.515,Z 305.827,A -85,B 0,C 180,E1 -14734.236,E2 -14734.236} C_VEL
LIN {X 0,Y 335.346,Z 321.984,A -85,B 0,C 180,E1 -14735.219,E2 -14735.219} C_VEL
LIN {X 0,Y 334.032,Z 337.492,A -85,B 0,C 180,E1 -14736.436,E2 -14736.436} C_VEL
LIN {X 0,Y 332.65,Z 351.599,A -85,B 0,C 180,E1 -14737.811,E2 -14737.811} C_VEL
LIN {X 0,Y 331.31,Z 364.594,A -85,B 0,C 180,E1 -14739.349,E2 -14739.349} C_VEL
LIN {X 0,Y 329.956,Z 376.575,A -85,B 0,C 180,E1 -14741.045,E2 -14741.045} C_VEL
LIN {X 0,Y 328.761,Z 387.605,A -85,B 0,C 180,E1 -14742.906,E2 -14742.906} C_VEL
LIN {X 0,Y 327.684,Z 397.194,A -85,B 0,C 180,E1 -14744.827,E2 -14744.827} C_VEL
LIN {X 0,Y 326.907,Z 406.088,A -85,B 0,C 180,E1 -14746.954,E2 -14746.954} C_VEL
LIN {X 0,Y 326.158,Z 412.674,A -85,B 0,C 180,E1 -14748.817,E2 -14748.817} C_VEL
LIN {X 0,Y 325.65,Z 419.878,A -85,B 0,C 180,E1 -14751.311,E2 -14751.311} C_VEL
LIN {X 0,Y 325.301,Z 425.485,A -85,B 0,C 180,E1 -14753.798,E2 -14753.798} C_VEL
LIN {X 0,Y 325.17,Z 429.64,A -85,B 0,C 180,E1 -14756.282,E2 -14756.282} C_VEL
LIN {X 0,Y 325.103,Z 432.462,A -85,B 0,C 180,E1 -14758.761,E2 -14758.761} C_VEL
LIN {X 0,Y 325.241,Z 434.017,A -85,B 0,C 180,E1 -14761.238,E2 -14761.238} C_VEL
LIN {X 0,Y 325.517,Z 434.315,A -85,B 0,C 180,E1 -14763.713,E2 -14763.713} C_VEL
LIN {X 0,Y 325.76,Z 433.369,A -85,B 0,C 180,E1 -14766.192,E2 -14766.192} C_VEL
LIN {X 0,Y 326.572,Z 431.17,A -85,B 0,C 180,E1 -14768.664,E2 -14768.664} C_VEL
LIN {X 0,Y 327.605,Z 427.721,A -85,B 0,C 180,E1 -14771.132,E2 -14771.132} C_VEL
LIN {X 0,Y 328.938,Z 422.961,A -85,B 0,C 180,E1 -14773.593,E2 -14773.593} C_VEL
LIN {X 0,Y 330.603,Z 416.798,A -85,B 0,C 180,E1 -14776.042,E2 -14776.042} C_VEL
LIN {X 0,Y 333.016,Z 408.998,A -85,B 0,C 180,E1 -14778.455,E2 -14778.455} C_VEL
LIN {X 0,Y 335.365,Z 400.733,A -85,B 0,C 180,E1 -14780.549,E2 -14780.549} C_VEL
LIN {X 0,Y 337.691,Z 392.408,A -85,B 0,C 180,E1 -14782.322,E2 -14782.322} C_VEL
LIN {X 0,Y 340.362,Z 382.689,A -85,B 0,C 180,E1 -14784.067,E2 -14784.067} C_VEL
LIN {X 0,Y 343.463,Z 370.598,A -85,B 0,C 180,E1 -14785.879,E2 -14785.879} C_VEL
LIN {X 0,Y 346.52,Z 357.744,A -85,B 0,C 180,E1 -14787.478,E2 -14787.478} C_VEL
LIN {X 0,Y 349.763,Z 342.795,A -85,B 0,C 180,E1 -14788.996,E2 -14788.996} C_VEL
LIN {X 0,Y 352.647,Z 327.901,A -85,B 0,C 180,E1 -14790.213,E2 -14790.213} C_VEL
LIN {X 0,Y 355.305,Z 311.987,A -85,B 0,C 180,E1 -14791.234,E2 -14791.234} C_VEL
LIN {X 0,Y 357.501,Z 295.909,A -85,B 0,C 180,E1 -14792.019,E2 -14792.019} C_VEL
LIN {X 0,Y 367.216,Z 223.442,A -85,B 0,C 180,E1 -14794.67,E2 -14794.67} C_VEL
LIN {X 0,Y 371.738,Z 193.704,A -85,B 0,C 180,E1 -14795.759,E2 -14795.759} C_VEL
LIN {X 0,Y 369.067,Z 188.601,A -85,B 0,C 180,E1 -14797.187,E2 -14797.187} C_VEL
LIN {X 0,Y 366.88,Z 185.182,A -85,B 0,C 180,E1 -14798.546,E2 -14798.546} C_VEL
LIN {X 0,Y 365.269,Z 182.872,A -85,B 0,C 180,E1 -14799.791,E2 -14799.791} C_VEL
LIN {X 0,Y 363.36,Z 180.433,A -85,B 0,C 180,E1 -14801.936,E2 -14801.936} C_VEL
LIN {X 0,Y 362.361,Z 180.513,A -85,B 0,C 180,E1 -14804.284,E2 -14804.284} C_VEL
LIN {X 0,Y 362.52,Z 181.885,A -85,B 0,C 180,E1 -14806.152,E2 -14806.152} C_VEL
LIN {X 0,Y 363.884,Z 185.351,A -85,B 0,C 180,E1 -14808.474,E2 -14808.474} C_VEL
LIN {X 0,Y 366.204,Z 191.776,A -85,B 0,C 180,E1 -14810.742,E2 -14810.742} C_VEL
LIN {X 0,Y 368.193,Z 197.505,A -85,B 0,C 180,E1 -14812.173,E2 -14812.173} C_VEL
LIN {X 0,Y 369.497,Z 201.837,A -85,B 0,C 180,E1 -14813.021,E2 -14813.021} C_VEL
LIN {X 0,Y 369.438,Z 214.664,A -85,B 0,C 180,E1 -14814.072,E2 -14814.072} C_VEL
LIN {X 0,Y 368.304,Z 223.056,A -85,B 0,C 180,E1 -14814.399,E2 -14814.399} C_VEL
LIN {X 0,Y 359.404,Z 288.833,A -85,B 0,C 180,E1 -14816.76,E2 -14816.76} C_VEL
LIN {X 0,Y 355.126,Z 323.332,A -85,B 0,C 180,E1 -14818.036,E2 -14818.036} C_VEL
LIN {X 0,Y 352.142,Z 341.115,A -85,B 0,C 180,E1 -14818.908,E2 -14818.908} C_VEL
LIN {X 0,Y 348.928,Z 357.094,A -85,B 0,C 180,E1 -14819.932,E2 -14819.932} C_VEL
LIN {X 0,Y 345.716,Z 371.866,A -85,B 0,C 180,E1 -14821.134,E2 -14821.134} C_VEL
LIN {X 0,Y 342.168,Z 386.892,A -85,B 0,C 180,E1 -14822.64,E2 -14822.64} C_VEL
LIN {X 0,Y 338.76,Z 400.71,A -85,B 0,C 180,E1 -14824.337,E2 -14824.337} C_VEL
LIN {X 0,Y 335.608,Z 413.385,A -85,B 0,C 180,E1 -14826.227,E2 -14826.227} C_VEL
LIN {X 0,Y 332.827,Z 424.855,A -85,B 0,C 180,E1 -14828.295,E2 -14828.295} C_VEL
LIN {X 0,Y 330.438,Z 434.735,A -85,B 0,C 180,E1 -14830.429,E2 -14830.429} C_VEL
LIN {X 0,Y 328.185,Z 446.037,A -85,B 0,C 180,E1 -14833.196,E2 -14833.196} C_VEL
LIN {X 0,Y 326.798,Z 454.056,A -85,B 0,C 180,E1 -14835.593,E2 -14835.593} C_VEL
LIN {X 0,Y 325.813,Z 460.927,A -85,B 0,C 180,E1 -14838.175,E2 -14838.175} C_VEL
LIN {X 0,Y 325.203,Z 466.076,A -85,B 0,C 180,E1 -14840.672,E2 -14840.672} C_VEL
LIN {X 0,Y 325.011,Z 469.055,A -85,B 0,C 180,E1 -14842.545,E2 -14842.545} C_VEL
LIN {X 0,Y 324.872,Z 471.9,A -85,B 0,C 180,E1 -14845.036,E2 -14845.036} C_VEL
LIN {X 0,Y 324.87,Z 473.531,A -85,B 0,C 180,E1 -14847.52,E2 -14847.52} C_VEL
LIN {X 0,Y 324.877,Z 473.971,A -85,B 0,C 180,E1 -14850,E2 -14850} C_VEL
LIN {X 0,Y 324.872,Z 473.222,A -85,B 0,C 180,E1 -14852.48,E2 -14852.48} C_VEL
LIN {X 0,Y 324.881,Z 471.259,A -85,B 0,C 180,E1 -14854.964,E2 -14854.964} C_VEL
LIN {X 0,Y 325.032,Z 468.011,A -85,B 0,C 180,E1 -14857.454,E2 -14857.454} C_VEL
LIN {X 0,Y 325.266,Z 463.425,A -85,B 0,C 180,E1 -14859.954,E2 -14859.954} C_VEL
LIN {X 0,Y 325.936,Z 457.408,A -85,B 0,C 180,E1 -14862.452,E2 -14862.452} C_VEL
LIN {X 0,Y 326.843,Z 449.774,A -85,B 0,C 180,E1 -14864.953,E2 -14864.953} C_VEL
LIN {X 0,Y 329.459,Z 436.595,A -85,B 0,C 180,E1 -14868.662,E2 -14868.662} C_VEL
LIN {X 0,Y 331.496,Z 427.327,A -85,B 0,C 180,E1 -14870.8,E2 -14870.8} C_VEL
LIN {X 0,Y 334.088,Z 416.442,A -85,B 0,C 180,E1 -14872.903,E2 -14872.903} C_VEL
LIN {X 0,Y 337.38,Z 403.449,A -85,B 0,C 180,E1 -14874.95,E2 -14874.95} C_VEL
LIN {X 0,Y 340.561,Z 390.281,A -85,B 0,C 180,E1 -14876.67,E2 -14876.67} C_VEL
LIN {X 0,Y 344.036,Z 375.54,A -85,B 0,C 180,E1 -14878.229,E2 -14878.229} C_VEL
LIN {X 0,Y 346.967,Z 361.873,A -85,B 0,C 180,E1 -14879.427,E2 -14879.427} C_VEL
LIN {X 0,Y 350.404,Z 344.915,A -85,B 0,C 180,E1 -14880.593,E2 -14880.593} C_VEL
LIN {X 0,Y 353.318,Z 328.229,A -85,B 0,C 180,E1 -14881.477,E2 -14881.477} C_VEL
LIN {X 0,Y 356.102,Z 307.599,A -85,B 0,C 180,E1 -14882.283,E2 -14882.283} C_VEL
LIN {X 0,Y 364.695,Z 239.836,A -85,B 0,C 180,E1 -14884.729,E2 -14884.729} C_VEL
LIN {X 0,Y 369.033,Z 209.34,A -85,B 0,C 180,E1 -14885.855,E2 -14885.855} C_VEL
LIN {X 0,Y 369.915,Z 193.981,A -85,B 0,C 180,E1 -14886.874,E2 -14886.874} C_VEL
LIN {X 0,Y 369.715,Z 191.623,A -85,B 0,C 180,E1 -14887.146,E2 -14887.146} C_VEL
LIN {X 0,Y 368.771,Z 185.232,A -85,B 0,C 180,E1 -14888.104,E2 -14888.104} C_VEL
LIN {X 0,Y 366.04,Z 180.047,A -85,B 0,C 180,E1 -14889.928,E2 -14889.928} C_VEL
LIN {X 0,Y 363.841,Z 176.065,A -85,B 0,C 180,E1 -14892.047,E2 -14892.047} C_VEL
LIN {X 0,Y 362.425,Z 174.328,A -85,B 0,C 180,E1 -14894.636,E2 -14894.636} C_VEL
LIN {X 0,Y 362.508,Z 174.308,A -85,B 0,C 180,E1 -14896.655,E2 -14896.655} C_VEL
LIN {X 0,Y 363.851,Z 175.84,A -85,B 0,C 180,E1 -14898.949,E2 -14898.949} C_VEL
LIN {X 0,Y 364.634,Z 177.24,A -85,B 0,C 180,E1 -14899.821,E2 -14899.821} C_VEL
LIN {X 0,Y 366.59,Z 180.544,A -85,B 0,C 180,E1 -14901.461,E2 -14901.461} C_VEL
LIN {X 0,Y 368.531,Z 184.262,A -85,B 0,C 180,E1 -14902.736,E2 -14902.736} C_VEL
LIN {X 0,Y 370.942,Z 189.154,A -85,B 0,C 180,E1 -14904.061,E2 -14904.061} C_VEL
LIN {X 0,Y 371.479,Z 190.51,A -85,B 0,C 180,E1 -14904.347,E2 -14904.347} C_VEL
LIN {X 0,Y 360.254,Z 269.286,A -85,B 0,C 180,E1 -14907.195,E2 -14907.195} C_VEL
LIN {X 0,Y 356.805,Z 297.212,A -85,B 0,C 180,E1 -14908.223,E2 -14908.223} C_VEL
LIN {X 0,Y 354.715,Z 312.593,A -85,B 0,C 180,E1 -14908.994,E2 -14908.994} C_VEL
LIN {X 0,Y 352.321,Z 327.056,A -85,B 0,C 180,E1 -14909.922,E2 -14909.922} C_VEL
LIN {X 0,Y 349.45,Z 342.152,A -85,B 0,C 180,E1 -14911.14,E2 -14911.14} C_VEL
LIN {X 0,Y 346.293,Z 357.111,A -85,B 0,C 180,E1 -14912.667,E2 -14912.667} C_VEL
LIN {X 0,Y 343.141,Z 370.403,A -85,B 0,C 180,E1 -14914.314,E2 -14914.314} C_VEL
LIN {X 0,Y 339.805,Z 383.103,A -85,B 0,C 180,E1 -14916.215,E2 -14916.215} C_VEL
LIN {X 0,Y 336.848,Z 394.208,A -85,B 0,C 180,E1 -14918.264,E2 -14918.264} C_VEL
LIN {X 0,Y 334.358,Z 403.461,A -85,B 0,C 180,E1 -14920.348,E2 -14920.348} C_VEL
LIN {X 0,Y 331.786,Z 412.214,A -85,B 0,C 180,E1 -14922.75,E2 -14922.75} C_VEL
LIN {X 0,Y 330.11,Z 417.675,A -85,B 0,C 180,E1 -14924.567,E2 -14924.567} C_VEL
LIN {X 0,Y 328.475,Z 423.584,A -85,B 0,C 180,E1 -14927.018,E2 -14927.018} C_VEL
LIN {X 0,Y 327.581,Z 427.076,A -85,B 0,C 180,E1 -14928.867,E2 -14928.867} C_VEL
LIN {X 0,Y 326.531,Z 430.6,A -85,B 0,C 180,E1 -14931.335,E2 -14931.335} C_VEL
LIN {X 0,Y 325.733,Z 432.867,A -85,B 0,C 180,E1 -14933.807,E2 -14933.807} C_VEL
LIN {X 0,Y 325.47,Z 433.865,A -85,B 0,C 180,E1 -14936.286,E2 -14936.286} C_VEL
LIN {X 0,Y 325.2,Z 433.62,A -85,B 0,C 180,E1 -14938.762,E2 -14938.762} C_VEL
LIN {X 0,Y 325.08,Z 432.128,A -85,B 0,C 180,E1 -14941.239,E2 -14941.239} C_VEL
LIN {X 0,Y 325.138,Z 429.36,A -85,B 0,C 180,E1 -14943.718,E2 -14943.718} C_VEL
LIN {X 0,Y 325.301,Z 425.248,A -85,B 0,C 180,E1 -14946.202,E2 -14946.202} C_VEL
LIN {X 0,Y 325.631,Z 419.692,A -85,B 0,C 180,E1 -14948.69,E2 -14948.69} C_VEL
LIN {X 0,Y 326.126,Z 412.546,A -85,B 0,C 180,E1 -14951.184,E2 -14951.184} C_VEL
LIN {X 0,Y 326.939,Z 404.8,A -85,B 0,C 180,E1 -14953.361,E2 -14953.361} C_VEL
LIN {X 0,Y 327.778,Z 395.437,A -85,B 0,C 180,E1 -14955.546,E2 -14955.546} C_VEL
LIN {X 0,Y 329.027,Z 384.153,A -85,B 0,C 180,E1 -14957.721,E2 -14957.721} C_VEL
LIN {X 0,Y 330.351,Z 372.51,A -85,B 0,C 180,E1 -14959.577,E2 -14959.577} C_VEL
LIN {X 0,Y 331.687,Z 359.756,A -85,B 0,C 180,E1 -14961.276,E2 -14961.276} C_VEL
LIN {X 0,Y 333.141,Z 345.829,A -85,B 0,C 180,E1 -14962.808,E2 -14962.808} C_VEL
LIN {X 0,Y 334.552,Z 330.443,A -85,B 0,C 180,E1 -14964.183,E2 -14964.183} C_VEL
LIN {X 0,Y 335.801,Z 315.476,A -85,B 0,C 180,E1 -14965.242,E2 -14965.242} C_VEL
LIN {X 0,Y 336.777,Z 299.578,A -85,B 0,C 180,E1 -14966.113,E2 -14966.113} C_VEL
LIN {X 0,Y 337.571,Z 283.646,A -85,B 0,C 180,E1 -14966.737,E2 -14966.737} C_VEL
LIN {X 0,Y 342.731,Z 168.769,A -85,B 0,C 180,E1 -14970.053,E2 -14970.053} C_VEL
LIN {X 0,Y 338.891,Z 159.407,A -85,B 0,C 180,E1 -14970.612,E2 -14970.612} C_VEL
LIN {X 0,Y 326.681,Z 130.906,A -85,B 0,C 180,E1 -14972.427,E2 -14972.427} C_VEL
LIN {X 0,Y 326.624,Z 130.425,A -85,B 0,C 180,E1 -14972.481,E2 -14972.481} C_VEL
LIN {X 0,Y 326.614,Z 130.426,A -85,B 0,C 180,E1 -14975.52,E2 -14975.52} C_VEL
LIN {X 0,Y 326.59,Z 130.43,A -85,B 0,C 180,E1 -14979.222,E2 -14979.222} C_VEL
LIN {X 0,Y 326.575,Z 130.431,A -85,B 0,C 180,E1 -14982.972,E2 -14982.972} C_VEL
LIN {X 0,Y 326.574,Z 130.399,A -85,B 0,C 180,E1 -14987.029,E2 -14987.029} C_VEL
LIN {X 0,Y 326.584,Z 130.428,A -85,B 0,C 180,E1 -14991.386,E2 -14991.386} C_VEL
LIN {X 0,Y 326.62,Z 130.401,A -85,B 0,C 180,E1 -14994.852,E2 -14994.852} C_VEL
LIN {X 0,Y 326.61,Z 130.427,A -85,B 0,C 180,E1 -14997.456,E2 -14997.456} C_VEL
LIN {X 0,Y 326.618,Z 130.408,A -85,B 0,C 180,E1 -15000.337,E2 -15000.337} C_VEL
LIN {X 0,Y 326.603,Z 130.422,A -85,B 0,C 180,E1 -15004.509,E2 -15004.509} C_VEL
LIN {X 0,Y 326.613,Z 130.426,A -85,B 0,C 180,E1 -15008.543,E2 -15008.543} C_VEL
LIN {X 0,Y 326.651,Z 130.416,A -85,B 0,C 180,E1 -15011.206,E2 -15011.206} C_VEL
LIN {X 0,Y 326.728,Z 130.414,A -85,B 0,C 180,E1 -15015.459,E2 -15015.459} C_VEL
LIN {X 0,Y 326.788,Z 130.459,A -85,B 0,C 180,E1 -15019.349,E2 -15019.349} C_VEL
LIN {X 0,Y 331.121,Z 144.245,A -85,B 0,C 180,E1 -15022.377,E2 -15022.377} C_VEL
LIN {X 0,Y 331.565,Z 145.387,A -85,B 0,C 180,E1 -15022.538,E2 -15022.538} C_VEL
LIN {X 0,Y 342.463,Z 168.606,A -85,B 0,C 180,E1 -15024.25,E2 -15024.25} C_VEL
LIN {X 0,Y 346.955,Z 179.834,A -85,B 0,C 180,E1 -15024.961,E2 -15024.961} C_VEL
LIN {X 0,Y 347.997,Z 186.184,A -85,B 0,C 180,E1 -15025.214,E2 -15025.214} C_VEL
LIN {X 0,Y 344,Z 311.624,A -85,B 0,C 180,E1 -15027.878,E2 -15027.878} C_VEL
LIN {X 0,Y 343.022,Z 327.21,A -85,B 0,C 180,E1 -15028.422,E2 -15028.422} C_VEL
LIN {X 0,Y 341.793,Z 342.186,A -85,B 0,C 180,E1 -15029.19,E2 -15029.19} C_VEL
LIN {X 0,Y 340.271,Z 356.332,A -85,B 0,C 180,E1 -15030.148,E2 -15030.148} C_VEL
LIN {X 0,Y 338.706,Z 368.636,A -85,B 0,C 180,E1 -15031.189,E2 -15031.189} C_VEL
LIN {X 0,Y 336.782,Z 381.642,A -85,B 0,C 180,E1 -15032.542,E2 -15032.542} C_VEL
LIN {X 0,Y 334.876,Z 393.633,A -85,B 0,C 180,E1 -15034.062,E2 -15034.062} C_VEL
LIN {X 0,Y 332.965,Z 404.742,A -85,B 0,C 180,E1 -15035.754,E2 -15035.754} C_VEL
LIN {X 0,Y 331.134,Z 414.968,A -85,B 0,C 180,E1 -15037.623,E2 -15037.623} C_VEL
LIN {X 0,Y 329.288,Z 424.98,A -85,B 0,C 180,E1 -15039.831,E2 -15039.831} C_VEL
LIN {X 0,Y 327.874,Z 433.247,A -85,B 0,C 180,E1 -15042.063,E2 -15042.063} C_VEL
LIN {X 0,Y 326.764,Z 440.1,A -85,B 0,C 180,E1 -15044.337,E2 -15044.337} C_VEL
LIN {X 0,Y 325.748,Z 442.621,A -85,B 0,C 180,E1 -15045.258,E2 -15045.258} C_VEL
LIN {X 0,Y 320.995,Z 447.743,A -85,B 0,C 180,E1 -15047.387,E2 -15047.387} C_VEL
LIN {X 0,Y 318.718,Z 450.132,A -85,B 0,C 180,E1 -15048.681,E2 -15048.681} C_VEL
LIN {X 0,Y 318.21,Z 451.157,A -85,B 0,C 180,E1 -15049.363,E2 -15049.363} C_VEL
LIN {X 0,Y 317.698,Z 454.565,A -85,B 0,C 180,E1 -15052.09,E2 -15052.09} C_VEL
LIN {X 0,Y 317.506,Z 456.599,A -85,B 0,C 180,E1 -15054.87,E2 -15054.87} C_VEL
LIN {X 0,Y 317.473,Z 457.242,A -85,B 0,C 180,E1 -15057.703,E2 -15057.703} C_VEL
LIN {X 0,Y 317.631,Z 456.425,A -85,B 0,C 180,E1 -15060.591,E2 -15060.591} C_VEL
LIN {X 0,Y 317.865,Z 454.78,A -85,B 0,C 180,E1 -15062.84,E2 -15062.84} C_VEL
LIN {X 0,Y 318.41,Z 451.951,A -85,B 0,C 180,E1 -15065.246,E2 -15065.246} C_VEL
LIN {X 0,Y 319.196,Z 447.259,A -85,B 0,C 180,E1 -15068.061,E2 -15068.061} C_VEL
LIN {X 0,Y 320.181,Z 442.104,A -85,B 0,C 180,E1 -15070.381,E2 -15070.381} C_VEL
LIN {X 0,Y 321.664,Z 434.764,A -85,B 0,C 180,E1 -15073.001,E2 -15073.001} C_VEL
LIN {X 0,Y 323.514,Z 426.515,A -85,B 0,C 180,E1 -15075.354,E2 -15075.354} C_VEL
LIN {X 0,Y 325.672,Z 417.021,A -85,B 0,C 180,E1 -15077.565,E2 -15077.565} C_VEL
LIN {X 0,Y 327.857,Z 406.709,A -85,B 0,C 180,E1 -15079.551,E2 -15079.551} C_VEL
LIN {X 0,Y 330.365,Z 394.856,A -85,B 0,C 180,E1 -15081.426,E2 -15081.426} C_VEL
LIN {X 0,Y 332.581,Z 383.226,A -85,B 0,C 180,E1 -15082.942,E2 -15082.942} C_VEL
LIN {X 0,Y 334.858,Z 369.941,A -85,B 0,C 180,E1 -15084.366,E2 -15084.366} C_VEL
LIN {X 0,Y 337.089,Z 355.189,A -85,B 0,C 180,E1 -15085.622,E2 -15085.622} C_VEL
LIN {X 0,Y 338.907,Z 340.521,A -85,B 0,C 180,E1 -15086.582,E2 -15086.582} C_VEL
LIN {X 0,Y 340.272,Z 325.573,A -85,B 0,C 180,E1 -15087.315,E2 -15087.315} C_VEL
LIN {X 0,Y 341.295,Z 309.609,A -85,B 0,C 180,E1 -15087.836,E2 -15087.836} C_VEL
LIN {X 0,Y 344.925,Z 208.65,A -85,B 0,C 180,E1 -15090.053,E2 -15090.053} C_VEL
LIN {X 0,Y 344.512,Z 209.04,A -85,B 0,C 180,E1 -15090.092,E2 -15090.092} C_VEL
LIN {X 0,Y 341.215,Z 219.088,A -85,B 0,C 180,E1 -15090.226,E2 -15090.226} C_VEL
LIN {X 0,Y 338.46,Z 224.642,A -85,B 0,C 180,E1 -15090.416,E2 -15090.416} C_VEL
LIN {X 0,Y 336.736,Z 226.554,A -85,B 0,C 180,E1 -15090.58,E2 -15090.58} C_VEL
LIN {X 0,Y 335.343,Z 226.732,A -85,B 0,C 180,E1 -15090.752,E2 -15090.752} C_VEL
LIN {X 0,Y 334.224,Z 224.944,A -85,B 0,C 180,E1 -15090.947,E2 -15090.947} C_VEL
LIN {X 0,Y 333.669,Z 221.709,A -85,B 0,C 180,E1 -15091.11,E2 -15091.11} C_VEL
LIN {X 0,Y 330.564,Z 290.054,A -85,B 0,C 180,E1 -15093.188,E2 -15093.188} C_VEL
LIN {X 0,Y 329.68,Z 305.931,A -85,B 0,C 180,E1 -15093.916,E2 -15093.916} C_VEL
LIN {X 0,Y 328.468,Z 322.083,A -85,B 0,C 180,E1 -15094.918,E2 -15094.918} C_VEL
LIN {X 0,Y 327.218,Z 336.741,A -85,B 0,C 180,E1 -15096.083,E2 -15096.083} C_VEL
LIN {X 0,Y 325.778,Z 351.021,A -85,B 0,C 180,E1 -15097.485,E2 -15097.485} C_VEL
LIN {X 0,Y 324.37,Z 364.5,A -85,B 0,C 180,E1 -15099.098,E2 -15099.098} C_VEL
LIN {X 0,Y 323.012,Z 376.284,A -85,B 0,C 180,E1 -15100.786,E2 -15100.786} C_VEL
LIN {X 0,Y 321.66,Z 388.295,A -85,B 0,C 180,E1 -15102.844,E2 -15102.844} C_VEL
LIN {X 0,Y 320.516,Z 398.329,A -85,B 0,C 180,E1 -15104.91,E2 -15104.91} C_VEL
LIN {X 0,Y 319.641,Z 407.934,A -85,B 0,C 180,E1 -15107.298,E2 -15107.298} C_VEL
LIN {X 0,Y 318.969,Z 414.268,A -85,B 0,C 180,E1 -15109.205,E2 -15109.205} C_VEL
LIN {X 0,Y 318.488,Z 421.242,A -85,B 0,C 180,E1 -15111.753,E2 -15111.753} C_VEL
LIN {X 0,Y 318.166,Z 426.295,A -85,B 0,C 180,E1 -15114.115,E2 -15114.115} C_VEL
LIN {X 0,Y 318.093,Z 429.754,A -85,B 0,C 180,E1 -15116.199,E2 -15116.199} C_VEL
LIN {X 0,Y 318.009,Z 432.72,A -85,B 0,C 180,E1 -15118.733,E2 -15118.733} C_VEL
LIN {X 0,Y 318.153,Z 434.392,A -85,B 0,C 180,E1 -15121.265,E2 -15121.265} C_VEL
LIN {X 0,Y 318.435,Z 434.805,A -85,B 0,C 180,E1 -15123.796,E2 -15123.796} C_VEL
LIN {X 0,Y 318.738,Z 434.005,A -85,B 0,C 180,E1 -15126.329,E2 -15126.329} C_VEL
LIN {X 0,Y 319.585,Z 431.965,A -85,B 0,C 180,E1 -15128.855,E2 -15128.855} C_VEL
LIN {X 0,Y 320.699,Z 428.68,A -85,B 0,C 180,E1 -15131.375,E2 -15131.375} C_VEL
LIN {X 0,Y 321.636,Z 425.397,A -85,B 0,C 180,E1 -15133.263,E2 -15133.263} C_VEL
LIN {X 0,Y 323.417,Z 419.778,A -85,B 0,C 180,E1 -15135.761,E2 -15135.761} C_VEL
LIN {X 0,Y 325.485,Z 413.595,A -85,B 0,C 180,E1 -15137.921,E2 -15137.921} C_VEL
LIN {X 0,Y 328.213,Z 405.005,A -85,B 0,C 180,E1 -15140.362,E2 -15140.362} C_VEL
LIN {X 0,Y 330.955,Z 395.931,A -85,B 0,C 180,E1 -15142.472,E2 -15142.472} C_VEL
LIN {X 0,Y 334.217,Z 385.091,A -85,B 0,C 180,E1 -15144.538,E2 -15144.538} C_VEL
LIN {X 0,Y 337.804,Z 372.296,A -85,B 0,C 180,E1 -15146.541,E2 -15146.541} C_VEL
LIN {X 0,Y 341.013,Z 359.977,A -85,B 0,C 180,E1 -15148.127,E2 -15148.127} C_VEL
LIN {X 0,Y 344.439,Z 345.519,A -85,B 0,C 180,E1 -15149.656,E2 -15149.656} C_VEL
LIN {X 0,Y 347.443,Z 331.3,A -85,B 0,C 180,E1 -15150.882,E2 -15150.882} C_VEL
LIN {X 0,Y 350.479,Z 315.15,A -85,B 0,C 180,E1 -15151.979,E2 -15151.979} C_VEL
LIN {X 0,Y 352.935,Z 299.21,A -85,B 0,C 180,E1 -15152.82,E2 -15152.82} C_VEL
LIN {X 0,Y 362.806,Z 230.454,A -85,B 0,C 180,E1 -15155.402,E2 -15155.402} C_VEL
LIN {X 0,Y 368.115,Z 197.995,A -85,B 0,C 180,E1 -15156.595,E2 -15156.595} C_VEL
LIN {X 0,Y 366.107,Z 194.18,A -85,B 0,C 180,E1 -15157.794,E2 -15157.794} C_VEL
LIN {X 0,Y 364.535,Z 191.57,A -85,B 0,C 180,E1 -15158.881,E2 -15158.881} C_VEL
LIN {X 0,Y 363.275,Z 189.601,A -85,B 0,C 180,E1 -15159.931,E2 -15159.931} C_VEL
LIN {X 0,Y 361.561,Z 187.318,A -85,B 0,C 180,E1 -15161.93,E2 -15161.93} C_VEL
LIN {X 0,Y 360.579,Z 187.348,A -85,B 0,C 180,E1 -15164.153,E2 -15164.153} C_VEL
LIN {X 0,Y 360.692,Z 188.821,A -85,B 0,C 180,E1 -15166.131,E2 -15166.131} C_VEL
LIN {X 0,Y 361.81,Z 192.055,A -85,B 0,C 180,E1 -15168.239,E2 -15168.239} C_VEL
LIN {X 0,Y 363.689,Z 197.84,A -85,B 0,C 180,E1 -15170.307,E2 -15170.307} C_VEL
LIN {X 0,Y 365.375,Z 203.195,A -85,B 0,C 180,E1 -15171.68,E2 -15171.68} C_VEL
LIN {X 0,Y 366.168,Z 206.446,A -85,B 0,C 180,E1 -15172.311,E2 -15172.311} C_VEL
LIN {X 0,Y 365.881,Z 217.079,A -85,B 0,C 180,E1 -15173.192,E2 -15173.192} C_VEL
LIN {X 0,Y 355.237,Z 289.536,A -85,B 0,C 180,E1 -15175.849,E2 -15175.849} C_VEL
LIN {X 0,Y 350.723,Z 322.92,A -85,B 0,C 180,E1 -15177.117,E2 -15177.117} C_VEL
LIN {X 0,Y 347.713,Z 339.712,A -85,B 0,C 180,E1 -15177.956,E2 -15177.956} C_VEL
LIN {X 0,Y 344.695,Z 353.854,A -85,B 0,C 180,E1 -15178.844,E2 -15178.844} C_VEL
LIN {X 0,Y 341.202,Z 368.933,A -85,B 0,C 180,E1 -15180.034,E2 -15180.034} C_VEL
LIN {X 0,Y 337.414,Z 384.201,A -85,B 0,C 180,E1 -15181.545,E2 -15181.545} C_VEL
LIN {X 0,Y 333.654,Z 398.225,A -85,B 0,C 180,E1 -15183.241,E2 -15183.241} C_VEL
LIN {X 0,Y 330.293,Z 411.06,A -85,B 0,C 180,E1 -15185.15,E2 -15185.15} C_VEL
LIN {X 0,Y 327.481,Z 421.287,A -85,B 0,C 180,E1 -15186.942,E2 -15186.942} C_VEL
LIN {X 0,Y 324.831,Z 431.496,A -85,B 0,C 180,E1 -15189.084,E2 -15189.084} C_VEL
LIN {X 0,Y 322.593,Z 440.197,A -85,B 0,C 180,E1 -15191.256,E2 -15191.256} C_VEL
LIN {X 0,Y 320.511,Z 450.353,A -85,B 0,C 180,E1 -15194.092,E2 -15194.092} C_VEL
LIN {X 0,Y 319.25,Z 457.742,A -85,B 0,C 180,E1 -15196.635,E2 -15196.635} C_VEL
LIN {X 0,Y 318.384,Z 463.579,A -85,B 0,C 180,E1 -15199.186,E2 -15199.186} C_VEL
LIN {X 0,Y 318.069,Z 467.049,A -85,B 0,C 180,E1 -15201.102,E2 -15201.102} C_VEL
LIN {X 0,Y 317.873,Z 470.494,A -85,B 0,C 180,E1 -15203.653,E2 -15203.653} C_VEL
LIN {X 0,Y 317.801,Z 472.704,A -85,B 0,C 180,E1 -15206.196,E2 -15206.196} C_VEL
LIN {X 0,Y 317.76,Z 473.718,A -85,B 0,C 180,E1 -15208.733,E2 -15208.733} C_VEL
LIN {X 0,Y 317.761,Z 473.544,A -85,B 0,C 180,E1 -15211.267,E2 -15211.267} C_VEL
LIN {X 0,Y 317.808,Z 472.174,A -85,B 0,C 180,E1 -15213.804,E2 -15213.804} C_VEL
LIN {X 0,Y 317.876,Z 469.561,A -85,B 0,C 180,E1 -15216.347,E2 -15216.347} C_VEL
LIN {X 0,Y 318.039,Z 465.63,A -85,B 0,C 180,E1 -15218.899,E2 -15218.899} C_VEL
LIN {X 0,Y 318.507,Z 460.32,A -85,B 0,C 180,E1 -15221.454,E2 -15221.454} C_VEL
LIN {X 0,Y 319.374,Z 453.495,A -85,B 0,C 180,E1 -15224.008,E2 -15224.008} C_VEL
LIN {X 0,Y 321.903,Z 440.591,A -85,B 0,C 180,E1 -15228.127,E2 -15228.127} C_VEL
LIN {X 0,Y 324.26,Z 430.95,A -85,B 0,C 180,E1 -15230.615,E2 -15230.615} C_VEL
LIN {X 0,Y 326.776,Z 420.792,A -85,B 0,C 180,E1 -15232.776,E2 -15232.776} C_VEL
LIN {X 0,Y 329.577,Z 410.676,A -85,B 0,C 180,E1 -15234.571,E2 -15234.571} C_VEL
LIN {X 0,Y 332.971,Z 397.845,A -85,B 0,C 180,E1 -15236.48,E2 -15236.48} C_VEL
LIN {X 0,Y 336.62,Z 383.897,A -85,B 0,C 180,E1 -15238.188,E2 -15238.188} C_VEL
LIN {X 0,Y 340.762,Z 366.854,A -85,B 0,C 180,E1 -15239.856,E2 -15239.856} C_VEL
LIN {X 0,Y 344.231,Z 351.523,A -85,B 0,C 180,E1 -15241.032,E2 -15241.032} C_VEL
LIN {X 0,Y 347.422,Z 335.791,A -85,B 0,C 180,E1 -15241.988,E2 -15241.988} C_VEL
LIN {X 0,Y 350.268,Z 319.196,A -85,B 0,C 180,E1 -15242.76,E2 -15242.76} C_VEL
LIN {X 0,Y 361.44,Z 237.735,A -85,B 0,C 180,E1 -15245.783,E2 -15245.783} C_VEL
LIN {X 0,Y 365.555,Z 210.935,A -85,B 0,C 180,E1 -15246.79,E2 -15246.79} C_VEL
LIN {X 0,Y 366.619,Z 196.728,A -85,B 0,C 180,E1 -15247.759,E2 -15247.759} C_VEL
LIN {X 0,Y 365.88,Z 190.777,A -85,B 0,C 180,E1 -15248.673,E2 -15248.673} C_VEL
LIN {X 0,Y 363.504,Z 186.088,A -85,B 0,C 180,E1 -15250.473,E2 -15250.473} C_VEL
LIN {X 0,Y 361.818,Z 182.712,A -85,B 0,C 180,E1 -15252.334,E2 -15252.334} C_VEL
LIN {X 0,Y 360.665,Z 181.247,A -85,B 0,C 180,E1 -15254.548,E2 -15254.548} C_VEL
LIN {X 0,Y 360.741,Z 181.194,A -85,B 0,C 180,E1 -15256.661,E2 -15256.661} C_VEL
LIN {X 0,Y 362.033,Z 182.745,A -85,B 0,C 180,E1 -15258.916,E2 -15258.916} C_VEL
LIN {X 0,Y 364.231,Z 186.762,A -85,B 0,C 180,E1 -15261.073,E2 -15261.073} C_VEL
LIN {X 0,Y 365.954,Z 190.351,A -85,B 0,C 180,E1 -15262.338,E2 -15262.338} C_VEL
LIN {X 0,Y 367.819,Z 194.525,A -85,B 0,C 180,E1 -15263.491,E2 -15263.491} C_VEL
LIN {X 0,Y 356.726,Z 266.707,A -85,B 0,C 180,E1 -15266.139,E2 -15266.139} C_VEL
LIN {X 0,Y 352.423,Z 298.627,A -85,B 0,C 180,E1 -15267.35,E2 -15267.35} C_VEL
LIN {X 0,Y 350.178,Z 313.619,A -85,B 0,C 180,E1 -15268.124,E2 -15268.124} C_VEL
LIN {X 0,Y 347.454,Z 328.706,A -85,B 0,C 180,E1 -15269.119,E2 -15269.119} C_VEL
LIN {X 0,Y 344.398,Z 343.382,A -85,B 0,C 180,E1 -15270.34,E2 -15270.34} C_VEL
LIN {X 0,Y 341.046,Z 358.074,A -85,B 0,C 180,E1 -15271.876,E2 -15271.876} C_VEL
LIN {X 0,Y 337.952,Z 370.252,A -85,B 0,C 180,E1 -15273.409,E2 -15273.409} C_VEL
LIN {X 0,Y 334.676,Z 381.97,A -85,B 0,C 180,E1 -15275.166,E2 -15275.166} C_VEL
LIN {X 0,Y 331.829,Z 391.775,A -85,B 0,C 180,E1 -15276.932,E2 -15276.932} C_VEL
LIN {X 0,Y 328.918,Z 401.477,A -85,B 0,C 180,E1 -15279.029,E2 -15279.029} C_VEL
LIN {X 0,Y 326.146,Z 410.644,A -85,B 0,C 180,E1 -15281.467,E2 -15281.467} C_VEL
LIN {X 0,Y 323.881,Z 417.282,A -85,B 0,C 180,E1 -15283.615,E2 -15283.615} C_VEL
LIN {X 0,Y 322.107,Z 423.347,A -85,B 0,C 180,E1 -15286.113,E2 -15286.113} C_VEL
LIN {X 0,Y 320.674,Z 428.016,A -85,B 0,C 180,E1 -15288.624,E2 -15288.624} C_VEL
LIN {X 0,Y 319.562,Z 431.375,A -85,B 0,C 180,E1 -15291.145,E2 -15291.145} C_VEL
LIN {X 0,Y 318.711,Z 433.487,A -85,B 0,C 180,E1 -15293.67,E2 -15293.67} C_VEL
LIN {X 0,Y 318.388,Z 434.355,A -85,B 0,C 180,E1 -15296.203,E2 -15296.203} C_VEL
LIN {X 0,Y 318.112,Z 433.997,A -85,B 0,C 180,E1 -15298.734,E2 -15298.734} C_VEL
LIN {X 0,Y 317.984,Z 432.374,A -85,B 0,C 180,E1 -15301.267,E2 -15301.267} C_VEL
LIN {X 0,Y 318.064,Z 429.459,A -85,B 0,C 180,E1 -15303.801,E2 -15303.801} C_VEL
LIN {X 0,Y 318.246,Z 425.073,A -85,B 0,C 180,E1 -15306.404,E2 -15306.404} C_VEL
LIN {X 0,Y 318.567,Z 419.476,A -85,B 0,C 180,E1 -15308.884,E2 -15308.884} C_VEL
LIN {X 0,Y 318.942,Z 414.104,A -85,B 0,C 180,E1 -15310.796,E2 -15310.796} C_VEL
LIN {X 0,Y 319.721,Z 406.602,A -85,B 0,C 180,E1 -15313.022,E2 -15313.022} C_VEL
LIN {X 0,Y 320.491,Z 397.491,A -85,B 0,C 180,E1 -15315.257,E2 -15315.257} C_VEL
LIN {X 0,Y 321.731,Z 386.525,A -85,B 0,C 180,E1 -15317.48,E2 -15317.48} C_VEL
LIN {X 0,Y 323.054,Z 375.271,A -85,B 0,C 180,E1 -15319.376,E2 -15319.376} C_VEL
LIN {X 0,Y 324.443,Z 362.274,A -85,B 0,C 180,E1 -15321.209,E2 -15321.209} C_VEL
LIN {X 0,Y 326,Z 348.261,A -85,B 0,C 180,E1 -15322.834,E2 -15322.834} C_VEL
LIN {X 0,Y 327.396,Z 333.335,A -85,B 0,C 180,E1 -15324.239,E2 -15324.239} C_VEL
LIN {X 0,Y 328.81,Z 317.895,A -85,B 0,C 180,E1 -15325.393,E2 -15325.393} C_VEL
LIN {X 0,Y 329.809,Z 301.706,A -85,B 0,C 180,E1 -15326.334,E2 -15326.334} C_VEL
LIN {X 0,Y 330.649,Z 285.892,A -85,B 0,C 180,E1 -15326.998,E2 -15326.998} C_VEL
LIN {X 0,Y 336.06,Z 170.174,A -85,B 0,C 180,E1 -15330.445,E2 -15330.445} C_VEL
LIN {X 0,Y 319.714,Z 131.976,A -85,B 0,C 180,E1 -15332.919,E2 -15332.919} C_VEL
LIN {X 0,Y 319.588,Z 131.301,A -85,B 0,C 180,E1 -15332.984,E2 -15332.984} C_VEL
LIN {X 0,Y 319.558,Z 131.303,A -85,B 0,C 180,E1 -15336.428,E2 -15336.428} C_VEL
LIN {X 0,Y 319.53,Z 131.309,A -85,B 0,C 180,E1 -15339.662,E2 -15339.662} C_VEL
LIN {X 0,Y 319.521,Z 131.305,A -85,B 0,C 180,E1 -15343.46,E2 -15343.46} C_VEL
LIN {X 0,Y 319.552,Z 131.273,A -85,B 0,C 180,E1 -15347.016,E2 -15347.016} C_VEL
LIN {X 0,Y 319.547,Z 131.305,A -85,B 0,C 180,E1 -15350.371,E2 -15350.371} C_VEL
LIN {X 0,Y 319.58,Z 131.276,A -85,B 0,C 180,E1 -15354.458,E2 -15354.458} C_VEL
LIN {X 0,Y 319.527,Z 131.308,A -85,B 0,C 180,E1 -15358.138,E2 -15358.138} C_VEL
LIN {X 0,Y 319.573,Z 131.29,A -85,B 0,C 180,E1 -15361.604,E2 -15361.604} C_VEL
LIN {X 0,Y 319.529,Z 131.294,A -85,B 0,C 180,E1 -15365.298,E2 -15365.298} C_VEL
LIN {X 0,Y 319.566,Z 131.304,A -85,B 0,C 180,E1 -15368.046,E2 -15368.046} C_VEL
LIN {X 0,Y 319.59,Z 131.302,A -85,B 0,C 180,E1 -15372.069,E2 -15372.069} C_VEL
LIN {X 0,Y 319.713,Z 131.285,A -85,B 0,C 180,E1 -15376.007,E2 -15376.007} C_VEL
LIN {X 0,Y 319.704,Z 131.303,A -85,B 0,C 180,E1 -15378.633,E2 -15378.633} C_VEL
LIN {X 0,Y 324.291,Z 145.245,A -85,B 0,C 180,E1 -15381.733,E2 -15381.733} C_VEL
LIN {X 0,Y 331.662,Z 160.69,A -85,B 0,C 180,E1 -15382.948,E2 -15382.948} C_VEL
LIN {X 0,Y 337.489,Z 173.453,A -85,B 0,C 180,E1 -15383.876,E2 -15383.876} C_VEL
LIN {X 0,Y 341.122,Z 182.705,A -85,B 0,C 180,E1 -15384.47,E2 -15384.47} C_VEL
LIN {X 0,Y 341.805,Z 186.382,A -85,B 0,C 180,E1 -15384.629,E2 -15384.629} C_VEL
LIN {X 0,Y 337.649,Z 312.277,A -85,B 0,C 180,E1 -15387.355,E2 -15387.355} C_VEL
LIN {X 0,Y 336.641,Z 327.666,A -85,B 0,C 180,E1 -15387.906,E2 -15387.906} C_VEL
LIN {X 0,Y 335.437,Z 341.967,A -85,B 0,C 180,E1 -15388.649,E2 -15388.649} C_VEL
LIN {X 0,Y 333.97,Z 355.271,A -85,B 0,C 180,E1 -15389.548,E2 -15389.548} C_VEL
LIN {X 0,Y 332.124,Z 369.333,A -85,B 0,C 180,E1 -15390.758,E2 -15390.758} C_VEL
LIN {X 0,Y 330.273,Z 381.305,A -85,B 0,C 180,E1 -15392.02,E2 -15392.02} C_VEL
LIN {X 0,Y 328.168,Z 394.183,A -85,B 0,C 180,E1 -15393.684,E2 -15393.684} C_VEL
LIN {X 0,Y 325.996,Z 406.148,A -85,B 0,C 180,E1 -15395.567,E2 -15395.567} C_VEL
LIN {X 0,Y 324.145,Z 416.194,A -85,B 0,C 180,E1 -15397.475,E2 -15397.475} C_VEL
LIN {X 0,Y 322.257,Z 426.008,A -85,B 0,C 180,E1 -15399.731,E2 -15399.731} C_VEL
LIN {X 0,Y 320.797,Z 434.14,A -85,B 0,C 180,E1 -15402.013,E2 -15402.013} C_VEL
LIN {X 0,Y 319.557,Z 441.56,A -85,B 0,C 180,E1 -15404.602,E2 -15404.602} C_VEL
LIN {X 0,Y 318.642,Z 447.618,A -85,B 0,C 180,E1 -15407.323,E2 -15407.323} C_VEL
LIN {X 0,Y 318.21,Z 451.157,A -85,B 0,C 180,E1 -15409.363,E2 -15409.363} C_VEL
LIN {X 0,Y 317.276,Z 452.619,A -85,B 0,C 180,E1 -15410.385,E2 -15410.385} C_VEL
LIN {X 0,Y 314.118,Z 454.652,A -85,B 0,C 180,E1 -15412.053,E2 -15412.053} C_VEL
LIN {X 0,Y 311.572,Z 455.89,A -85,B 0,C 180,E1 -15413.416,E2 -15413.416} C_VEL
LIN {X 0,Y 310.488,Z 456.574,A -85,B 0,C 180,E1 -15414.482,E2 -15414.482} C_VEL
LIN {X 0,Y 310.398,Z 456.736,A -85,B 0,C 180,E1 -15414.845,E2 -15414.845} C_VEL
LIN {X 0,Y 310.395,Z 457.405,A -85,B 0,C 180,E1 -15417.987,E2 -15417.987} C_VEL
LIN {X 0,Y 310.539,Z 456.637,A -85,B 0,C 180,E1 -15420.682,E2 -15420.682} C_VEL
LIN {X 0,Y 310.853,Z 454.789,A -85,B 0,C 180,E1 -15423.224,E2 -15423.224} C_VEL
LIN {X 0,Y 311.496,Z 451.562,A -85,B 0,C 180,E1 -15425.917,E2 -15425.917} C_VEL
LIN {X 0,Y 312.276,Z 447.273,A -85,B 0,C 180,E1 -15428.453,E2 -15428.453} C_VEL
LIN {X 0,Y 313.63,Z 440.702,A -85,B 0,C 180,E1 -15431.38,E2 -15431.38} C_VEL
LIN {X 0,Y 315.096,Z 433.944,A -85,B 0,C 180,E1 -15433.744,E2 -15433.744} C_VEL
LIN {X 0,Y 317.04,Z 425.668,A -85,B 0,C 180,E1 -15436.091,E2 -15436.091} C_VEL
LIN {X 0,Y 319.028,Z 417.375,A -85,B 0,C 180,E1 -15438.03,E2 -15438.03} C_VEL
LIN {X 0,Y 321.237,Z 407.522,A -85,B 0,C 180,E1 -15439.972,E2 -15439.972} C_VEL
LIN {X 0,Y 323.532,Z 397.029,A -85,B 0,C 180,E1 -15441.696,E2 -15441.696} C_VEL
LIN {X 0,Y 326.09,Z 384.492,A -85,B 0,C 180,E1 -15443.401,E2 -15443.401} C_VEL
LIN {X 0,Y 328.385,Z 372.009,A -85,B 0,C 180,E1 -15444.789,E2 -15444.789} C_VEL
LIN {X 0,Y 330.559,Z 358.421,A -85,B 0,C 180,E1 -15446.014,E2 -15446.014} C_VEL
LIN {X 0,Y 332.526,Z 343.919,A -85,B 0,C 180,E1 -15447.037,E2 -15447.037} C_VEL
LIN {X 0,Y 334.023,Z 329.055,A -85,B 0,C 180,E1 -15447.832,E2 -15447.832} C_VEL
LIN {X 0,Y 335.177,Z 313.993,A -85,B 0,C 180,E1 -15448.385,E2 -15448.385} C_VEL
LIN {X 0,Y 337.727,Z 248.268,A -85,B 0,C 180,E1 -15449.873,E2 -15449.873} C_VEL
LIN {X 0,Y 338.245,Z 233.151,A -85,B 0,C 180,E1 -15450.214,E2 -15450.214} C_VEL
LIN {X 0,Y 336.597,Z 233.853,A -85,B 0,C 180,E1 -15450.4,E2 -15450.4} C_VEL
LIN {X 0,Y 333.503,Z 243.363,A -85,B 0,C 180,E1 -15450.532,E2 -15450.532} C_VEL
LIN {X 0,Y 330.658,Z 249.366,A -85,B 0,C 180,E1 -15450.734,E2 -15450.734} C_VEL
LIN {X 0,Y 328.849,Z 251.483,A -85,B 0,C 180,E1 -15450.912,E2 -15450.912} C_VEL
LIN {X 0,Y 327.616,Z 251.725,A -85,B 0,C 180,E1 -15451.069,E2 -15451.069} C_VEL
LIN {X 0,Y 326.597,Z 250.663,A -85,B 0,C 180,E1 -15451.237,E2 -15451.237} C_VEL
LIN {X 0,Y 325.865,Z 247.294,A -85,B 0,C 180,E1 -15451.432,E2 -15451.432} C_VEL
LIN {X 0,Y 325.792,Z 246.462,A -85,B 0,C 180,E1 -15451.474,E2 -15451.474} C_VEL
LIN {X 0,Y 323.715,Z 291.028,A -85,B 0,C 180,E1 -15452.89,E2 -15452.89} C_VEL
LIN {X 0,Y 322.735,Z 307.375,A -85,B 0,C 180,E1 -15453.67,E2 -15453.67} C_VEL
LIN {X 0,Y 321.522,Z 323.148,A -85,B 0,C 180,E1 -15454.684,E2 -15454.684} C_VEL
LIN {X 0,Y 320.227,Z 337.659,A -85,B 0,C 180,E1 -15455.872,E2 -15455.872} C_VEL
LIN {X 0,Y 318.77,Z 351.833,A -85,B 0,C 180,E1 -15457.304,E2 -15457.304} C_VEL
LIN {X 0,Y 317.312,Z 365.442,A -85,B 0,C 180,E1 -15458.979,E2 -15458.979} C_VEL
LIN {X 0,Y 315.826,Z 377.987,A -85,B 0,C 180,E1 -15460.838,E2 -15460.838} C_VEL
LIN {X 0,Y 314.574,Z 388.936,A -85,B 0,C 180,E1 -15462.781,E2 -15462.781} C_VEL
LIN {X 0,Y 313.471,Z 398.302,A -85,B 0,C 180,E1 -15464.75,E2 -15464.75} C_VEL
LIN {X 0,Y 312.656,Z 407.315,A -85,B 0,C 180,E1 -15467.009,E2 -15467.009} C_VEL
LIN {X 0,Y 311.944,Z 413.854,A -85,B 0,C 180,E1 -15468.959,E2 -15468.959} C_VEL
LIN {X 0,Y 311.527,Z 419.42,A -85,B 0,C 180,E1 -15470.913,E2 -15470.913} C_VEL
LIN {X 0,Y 311.165,Z 425.363,A -85,B 0,C 180,E1 -15473.515,E2 -15473.515} C_VEL
LIN {X 0,Y 311.019,Z 429.82,A -85,B 0,C 180,E1 -15476.113,E2 -15476.113} C_VEL
LIN {X 0,Y 310.913,Z 432.915,A -85,B 0,C 180,E1 -15478.704,E2 -15478.704} C_VEL
LIN {X 0,Y 311.063,Z 434.726,A -85,B 0,C 180,E1 -15481.294,E2 -15481.294} C_VEL
LIN {X 0,Y 311.353,Z 435.294,A -85,B 0,C 180,E1 -15483.882,E2 -15483.882} C_VEL
LIN {X 0,Y 311.72,Z 434.654,A -85,B 0,C 180,E1 -15486.472,E2 -15486.472} C_VEL
LIN {X 0,Y 312.619,Z 432.78,A -85,B 0,C 180,E1 -15489.054,E2 -15489.054} C_VEL
LIN {X 0,Y 313.802,Z 429.671,A -85,B 0,C 180,E1 -15491.628,E2 -15491.628} C_VEL
LIN {X 0,Y 314.808,Z 426.495,A -85,B 0,C 180,E1 -15493.556,E2 -15493.556} C_VEL
LIN {X 0,Y 316.713,Z 421.08,A -85,B 0,C 180,E1 -15496.104,E2 -15496.104} C_VEL
LIN {X 0,Y 319.065,Z 414.705,A -85,B 0,C 180,E1 -15498.438,E2 -15498.438} C_VEL
LIN {X 0,Y 321.792,Z 406.798,A -85,B 0,C 180,E1 -15500.787,E2 -15500.787} C_VEL
LIN {X 0,Y 324.698,Z 398.026,A -85,B 0,C 180,E1 -15502.93,E2 -15502.93} C_VEL
LIN {X 0,Y 328.127,Z 387.551,A -85,B 0,C 180,E1 -15505.025,E2 -15505.025} C_VEL
LIN {X 0,Y 331.921,Z 375.23,A -85,B 0,C 180,E1 -15507.049,E2 -15507.049} C_VEL
LIN {X 0,Y 334.918,Z 364.62,A -85,B 0,C 180,E1 -15508.515,E2 -15508.515} C_VEL
LIN {X 0,Y 338.501,Z 351.173,A -85,B 0,C 180,E1 -15510.058,E2 -15510.058} C_VEL
LIN {X 0,Y 341.621,Z 338.15,A -85,B 0,C 180,E1 -15511.295,E2 -15511.295} C_VEL
LIN {X 0,Y 344.614,Z 324.306,A -85,B 0,C 180,E1 -15512.367,E2 -15512.367} C_VEL
LIN {X 0,Y 347.778,Z 307.201,A -85,B 0,C 180,E1 -15513.413,E2 -15513.413} C_VEL
LIN {X 0,Y 350.365,Z 290.128,A -85,B 0,C 180,E1 -15514.17,E2 -15514.17} C_VEL
LIN {X 0,Y 361.203,Z 222.038,A -85,B 0,C 180,E1 -15516.743,E2 -15516.743} C_VEL
LIN {X 0,Y 364.668,Z 202.428,A -85,B 0,C 180,E1 -15517.472,E2 -15517.472} C_VEL
LIN {X 0,Y 362.576,Z 198.449,A -85,B 0,C 180,E1 -15518.954,E2 -15518.954} C_VEL
LIN {X 0,Y 361.292,Z 196.363,A -85,B 0,C 180,E1 -15520.07,E2 -15520.07} C_VEL
LIN {X 0,Y 359.681,Z 194.146,A -85,B 0,C 180,E1 -15522.055,E2 -15522.055} C_VEL
LIN {X 0,Y 358.744,Z 194.34,A -85,B 0,C 180,E1 -15524.438,E2 -15524.438} C_VEL
LIN {X 0,Y 358.886,Z 195.906,A -85,B 0,C 180,E1 -15526.208,E2 -15526.208} C_VEL
LIN {X 0,Y 359.782,Z 198.846,A -85,B 0,C 180,E1 -15528.058,E2 -15528.058} C_VEL
LIN {X 0,Y 361.302,Z 204.151,A -85,B 0,C 180,E1 -15529.944,E2 -15529.944} C_VEL
LIN {X 0,Y 362.696,Z 209.223,A -85,B 0,C 180,E1 -15531.243,E2 -15531.243} C_VEL
LIN {X 0,Y 363.018,Z 210.761,A -85,B 0,C 180,E1 -15531.554,E2 -15531.554} C_VEL
LIN {X 0,Y 362.631,Z 218.734,A -85,B 0,C 180,E1 -15532.234,E2 -15532.234} C_VEL
LIN {X 0,Y 351.341,Z 290.14,A -85,B 0,C 180,E1 -15534.894,E2 -15534.894} C_VEL
LIN {X 0,Y 346.592,Z 322.461,A -85,B 0,C 180,E1 -15536.152,E2 -15536.152} C_VEL
LIN {X 0,Y 343.179,Z 340.041,A -85,B 0,C 180,E1 -15537.045,E2 -15537.045} C_VEL
LIN {X 0,Y 339.371,Z 356.415,A -85,B 0,C 180,E1 -15538.124,E2 -15538.124} C_VEL
LIN {X 0,Y 335.378,Z 372.185,A -85,B 0,C 180,E1 -15539.458,E2 -15539.458} C_VEL
LIN {X 0,Y 331.423,Z 386.698,A -85,B 0,C 180,E1 -15540.983,E2 -15540.983} C_VEL
LIN {X 0,Y 327.54,Z 400.149,A -85,B 0,C 180,E1 -15542.7,E2 -15542.7} C_VEL
LIN {X 0,Y 323.99,Z 412.533,A -85,B 0,C 180,E1 -15544.633,E2 -15544.633} C_VEL
LIN {X 0,Y 321.051,Z 422.388,A -85,B 0,C 180,E1 -15546.453,E2 -15546.453} C_VEL
LIN {X 0,Y 318.25,Z 432.286,A -85,B 0,C 180,E1 -15548.631,E2 -15548.631} C_VEL
LIN {X 0,Y 315.575,Z 441.814,A -85,B 0,C 180,E1 -15551.16,E2 -15551.16} C_VEL
LIN {X 0,Y 313.226,Z 452.346,A -85,B 0,C 180,E1 -15554.38,E2 -15554.38} C_VEL
LIN {X 0,Y 312.064,Z 459.303,A -85,B 0,C 180,E1 -15556.985,E2 -15556.985} C_VEL
LIN {X 0,Y 311.226,Z 464.744,A -85,B 0,C 180,E1 -15559.592,E2 -15559.592} C_VEL
LIN {X 0,Y 310.866,Z 468.81,A -85,B 0,C 180,E1 -15562.204,E2 -15562.204} C_VEL
LIN {X 0,Y 310.695,Z 471.605,A -85,B 0,C 180,E1 -15564.809,E2 -15564.809} C_VEL
LIN {X 0,Y 310.709,Z 473.191,A -85,B 0,C 180,E1 -15567.407,E2 -15567.407} C_VEL
LIN {X 0,Y 310.694,Z 473.588,A -85,B 0,C 180,E1 -15570,E2 -15570} C_VEL
LIN {X 0,Y 310.711,Z 472.794,A -85,B 0,C 180,E1 -15572.593,E2 -15572.593} C_VEL
LIN {X 0,Y 310.7,Z 470.787,A -85,B 0,C 180,E1 -15575.191,E2 -15575.191} C_VEL
LIN {X 0,Y 310.876,Z 467.506,A -85,B 0,C 180,E1 -15577.796,E2 -15577.796} C_VEL
LIN {X 0,Y 311.143,Z 462.867,A -85,B 0,C 180,E1 -15580.411,E2 -15580.411} C_VEL
LIN {X 0,Y 311.89,Z 456.789,A -85,B 0,C 180,E1 -15583.023,E2 -15583.023} C_VEL
LIN {X 0,Y 314.382,Z 444.202,A -85,B 0,C 180,E1 -15587.565,E2 -15587.565} C_VEL
LIN {X 0,Y 316.7,Z 435.463,A -85,B 0,C 180,E1 -15590.119,E2 -15590.119} C_VEL
LIN {X 0,Y 319.305,Z 425.893,A -85,B 0,C 180,E1 -15592.418,E2 -15592.418} C_VEL
LIN {X 0,Y 321.765,Z 417.205,A -85,B 0,C 180,E1 -15594.176,E2 -15594.176} C_VEL
LIN {X 0,Y 325.436,Z 404.775,A -85,B 0,C 180,E1 -15596.277,E2 -15596.277} C_VEL
LIN {X 0,Y 328.637,Z 393.342,A -85,B 0,C 180,E1 -15597.892,E2 -15597.892} C_VEL
LIN {X 0,Y 332.556,Z 379.494,A -85,B 0,C 180,E1 -15599.508,E2 -15599.508} C_VEL
LIN {X 0,Y 336.549,Z 363.836,A -85,B 0,C 180,E1 -15601.005,E2 -15601.005} C_VEL
LIN {X 0,Y 340.204,Z 348.748,A -85,B 0,C 180,E1 -15602.137,E2 -15602.137} C_VEL
LIN {X 0,Y 343.864,Z 331.474,A -85,B 0,C 180,E1 -15603.143,E2 -15603.143} C_VEL
LIN {X 0,Y 346.921,Z 313.471,A -85,B 0,C 180,E1 -15603.943,E2 -15603.943} C_VEL
LIN {X 0,Y 357.462,Z 242.309,A -85,B 0,C 180,E1 -15606.626,E2 -15606.626} C_VEL
LIN {X 0,Y 362.354,Z 212.568,A -85,B 0,C 180,E1 -15607.757,E2 -15607.757} C_VEL
LIN {X 0,Y 363.49,Z 200.358,A -85,B 0,C 180,E1 -15608.602,E2 -15608.602} C_VEL
LIN {X 0,Y 363.115,Z 196.293,A -85,B 0,C 180,E1 -15609.269,E2 -15609.269} C_VEL
LIN {X 0,Y 361.198,Z 192.407,A -85,B 0,C 180,E1 -15610.863,E2 -15610.863} C_VEL
LIN {X 0,Y 359.972,Z 189.547,A -85,B 0,C 180,E1 -15612.419,E2 -15612.419} C_VEL
LIN {X 0,Y 358.859,Z 188.06,A -85,B 0,C 180,E1 -15614.832,E2 -15614.832} C_VEL
LIN {X 0,Y 359.06,Z 188.164,A -85,B 0,C 180,E1 -15616.946,E2 -15616.946} C_VEL
LIN {X 0,Y 360.303,Z 189.813,A -85,B 0,C 180,E1 -15619.021,E2 -15619.021} C_VEL
LIN {X 0,Y 361.963,Z 193.254,A -85,B 0,C 180,E1 -15620.768,E2 -15620.768} C_VEL
LIN {X 0,Y 363.498,Z 196.666,A -85,B 0,C 180,E1 -15621.994,E2 -15621.994} C_VEL
LIN {X 0,Y 364.336,Z 198.676,A -85,B 0,C 180,E1 -15622.597,E2 -15622.597} C_VEL
LIN {X 0,Y 352.225,Z 272.858,A -85,B 0,C 180,E1 -15625.378,E2 -15625.378} C_VEL
LIN {X 0,Y 348.755,Z 297.023,A -85,B 0,C 180,E1 -15626.303,E2 -15626.303} C_VEL
LIN {X 0,Y 346.369,Z 311.776,A -85,B 0,C 180,E1 -15627.041,E2 -15627.041} C_VEL
LIN {X 0,Y 343.473,Z 327.032,A -85,B 0,C 180,E1 -15628.033,E2 -15628.033} C_VEL
LIN {X 0,Y 340.188,Z 341.946,A -85,B 0,C 180,E1 -15629.249,E2 -15629.249} C_VEL
LIN {X 0,Y 336.879,Z 355.637,A -85,B 0,C 180,E1 -15630.643,E2 -15630.643} C_VEL
LIN {X 0,Y 333.117,Z 369.425,A -85,B 0,C 180,E1 -15632.345,E2 -15632.345} C_VEL
LIN {X 0,Y 329.51,Z 381.656,A -85,B 0,C 180,E1 -15634.192,E2 -15634.192} C_VEL
LIN {X 0,Y 326.549,Z 391.029,A -85,B 0,C 180,E1 -15635.863,E2 -15635.863} C_VEL
LIN {X 0,Y 323.355,Z 400.873,A -85,B 0,C 180,E1 -15637.981,E2 -15637.981} C_VEL
LIN {X 0,Y 320.667,Z 409.135,A -85,B 0,C 180,E1 -15640.141,E2 -15640.141} C_VEL
LIN {X 0,Y 317.905,Z 416.946,A -85,B 0,C 180,E1 -15642.636,E2 -15642.636} C_VEL
LIN {X 0,Y 316.174,Z 421.776,A -85,B 0,C 180,E1 -15644.53,E2 -15644.53} C_VEL
LIN {X 0,Y 314.392,Z 426.935,A -85,B 0,C 180,E1 -15647.083,E2 -15647.083} C_VEL
LIN {X 0,Y 313.168,Z 430.732,A -85,B 0,C 180,E1 -15649.658,E2 -15649.658} C_VEL
LIN {X 0,Y 312.094,Z 433.299,A -85,B 0,C 180,E1 -15652.235,E2 -15652.235} C_VEL
LIN {X 0,Y 311.408,Z 434.633,A -85,B 0,C 180,E1 -15654.821,E2 -15654.821} C_VEL
LIN {X 0,Y 311.205,Z 434.727,A -85,B 0,C 180,E1 -15657.412,E2 -15657.412} C_VEL
LIN {X 0,Y 310.951,Z 433.598,A -85,B 0,C 180,E1 -15660,E2 -15660} C_VEL
LIN {X 0,Y 310.91,Z 431.204,A -85,B 0,C 180,E1 -15662.592,E2 -15662.592} C_VEL
LIN {X 0,Y 311.038,Z 427.479,A -85,B 0,C 180,E1 -15665.186,E2 -15665.186} C_VEL
LIN {X 0,Y 311.355,Z 422.337,A -85,B 0,C 180,E1 -15667.784,E2 -15667.784} C_VEL
LIN {X 0,Y 311.762,Z 415.631,A -85,B 0,C 180,E1 -15670.39,E2 -15670.39} C_VEL
LIN {X 0,Y 312.478,Z 408.352,A -85,B 0,C 180,E1 -15672.668,E2 -15672.668} C_VEL
LIN {X 0,Y 313.223,Z 399.967,A -85,B 0,C 180,E1 -15674.845,E2 -15674.845} C_VEL
LIN {X 0,Y 314.267,Z 390.515,A -85,B 0,C 180,E1 -15676.902,E2 -15676.902} C_VEL
LIN {X 0,Y 315.469,Z 379.901,A -85,B 0,C 180,E1 -15678.847,E2 -15678.847} C_VEL
LIN {X 0,Y 316.97,Z 367.269,A -85,B 0,C 180,E1 -15680.779,E2 -15680.779} C_VEL
LIN {X 0,Y 318.392,Z 354.722,A -85,B 0,C 180,E1 -15682.382,E2 -15682.382} C_VEL
LIN {X 0,Y 319.755,Z 341.191,A -85,B 0,C 180,E1 -15683.821,E2 -15683.821} C_VEL
LIN {X 0,Y 321.127,Z 326.509,A -85,B 0,C 180,E1 -15685.09,E2 -15685.09} C_VEL
LIN {X 0,Y 322.301,Z 312.037,A -85,B 0,C 180,E1 -15686.087,E2 -15686.087} C_VEL
LIN {X 0,Y 323.33,Z 295.231,A -85,B 0,C 180,E1 -15686.968,E2 -15686.968} C_VEL
LIN {X 0,Y 324.188,Z 277.566,A -85,B 0,C 180,E1 -15687.606,E2 -15687.606} C_VEL
LIN {X 0,Y 329.238,Z 171.677,A -85,B 0,C 180,E1 -15690.854,E2 -15690.854} C_VEL
LIN {X 0,Y 312.66,Z 132.903,A -85,B 0,C 180,E1 -15693.427,E2 -15693.427} C_VEL
LIN {X 0,Y 312.527,Z 132.182,A -85,B 0,C 180,E1 -15693.501,E2 -15693.501} C_VEL
LIN {X 0,Y 312.516,Z 132.183,A -85,B 0,C 180,E1 -15697.387,E2 -15697.387} C_VEL
LIN {X 0,Y 312.443,Z 132.19,A -85,B 0,C 180,E1 -15700.717,E2 -15700.717} C_VEL
LIN {X 0,Y 312.452,Z 132.181,A -85,B 0,C 180,E1 -15704.21,E2 -15704.21} C_VEL
LIN {X 0,Y 312.456,Z 132.165,A -85,B 0,C 180,E1 -15707.925,E2 -15707.925} C_VEL
LIN {X 0,Y 312.486,Z 132.181,A -85,B 0,C 180,E1 -15711.923,E2 -15711.923} C_VEL
LIN {X 0,Y 312.532,Z 132.153,A -85,B 0,C 180,E1 -15714.22,E2 -15714.22} C_VEL
LIN {X 0,Y 312.504,Z 132.185,A -85,B 0,C 180,E1 -15717.334,E2 -15717.334} C_VEL
LIN {X 0,Y 312.509,Z 132.167,A -85,B 0,C 180,E1 -15721.292,E2 -15721.292} C_VEL
LIN {X 0,Y 312.52,Z 132.172,A -85,B 0,C 180,E1 -15724.705,E2 -15724.705} C_VEL
LIN {X 0,Y 312.542,Z 132.178,A -85,B 0,C 180,E1 -15727.526,E2 -15727.526} C_VEL
LIN {X 0,Y 312.554,Z 132.177,A -85,B 0,C 180,E1 -15731.651,E2 -15731.651} C_VEL
LIN {X 0,Y 312.655,Z 132.167,A -85,B 0,C 180,E1 -15735.684,E2 -15735.684} C_VEL
LIN {X 0,Y 312.654,Z 132.329,A -85,B 0,C 180,E1 -15737.917,E2 -15737.917} C_VEL
LIN {X 0,Y 316.989,Z 145.296,A -85,B 0,C 180,E1 -15740.892,E2 -15740.892} C_VEL
LIN {X 0,Y 324.867,Z 161.248,A -85,B 0,C 180,E1 -15742.228,E2 -15742.228} C_VEL
LIN {X 0,Y 332.202,Z 177.503,A -85,B 0,C 180,E1 -15743.44,E2 -15743.44} C_VEL
LIN {X 0,Y 335.269,Z 185.442,A -85,B 0,C 180,E1 -15743.956,E2 -15743.956} C_VEL
LIN {X 0,Y 335.62,Z 188.846,A -85,B 0,C 180,E1 -15744.078,E2 -15744.078} C_VEL
LIN {X 0,Y 331.393,Z 311.748,A -85,B 0,C 180,E1 -15746.776,E2 -15746.776} C_VEL
LIN {X 0,Y 330.339,Z 327.254,A -85,B 0,C 180,E1 -15747.328,E2 -15747.328} C_VEL
LIN {X 0,Y 329.105,Z 341.758,A -85,B 0,C 180,E1 -15748.088,E2 -15748.088} C_VEL
LIN {X 0,Y 327.476,Z 356.078,A -85,B 0,C 180,E1 -15749.078,E2 -15749.078} C_VEL
LIN {X 0,Y 325.557,Z 370.035,A -85,B 0,C 180,E1 -15750.309,E2 -15750.309} C_VEL
LIN {X 0,Y 323.446,Z 383.353,A -85,B 0,C 180,E1 -15751.774,E2 -15751.774} C_VEL
LIN {X 0,Y 321.255,Z 395.795,A -85,B 0,C 180,E1 -15753.449,E2 -15753.449} C_VEL
LIN {X 0,Y 319.073,Z 407.388,A -85,B 0,C 180,E1 -15755.346,E2 -15755.346} C_VEL
LIN {X 0,Y 317.16,Z 417.383,A -85,B 0,C 180,E1 -15757.32,E2 -15757.32} C_VEL
LIN {X 0,Y 315.216,Z 427.039,A -85,B 0,C 180,E1 -15759.626,E2 -15759.626} C_VEL
LIN {X 0,Y 313.741,Z 435.02,A -85,B 0,C 180,E1 -15761.959,E2 -15761.959} C_VEL
LIN {X 0,Y 312.582,Z 441.605,A -85,B 0,C 180,E1 -15764.319,E2 -15764.319} C_VEL
LIN {X 0,Y 311.621,Z 447.601,A -85,B 0,C 180,E1 -15767.049,E2 -15767.049} C_VEL
LIN {X 0,Y 311.005,Z 452.124,A -85,B 0,C 180,E1 -15769.814,E2 -15769.814} C_VEL
LIN {X 0,Y 310.547,Z 455.262,A -85,B 0,C 180,E1 -15772.627,E2 -15772.627} C_VEL
LIN {X 0,Y 310.398,Z 456.736,A -85,B 0,C 180,E1 -15774.845,E2 -15774.845} C_VEL
LIN {X 0,Y 309.709,Z 457.214,A -85,B 0,C 180,E1 -15775.924,E2 -15775.924} C_VEL
LIN {X 0,Y 306.818,Z 457.536,A -85,B 0,C 180,E1 -15777.687,E2 -15777.687} C_VEL
LIN {X 0,Y 304.426,Z 457.438,A -85,B 0,C 180,E1 -15779.118,E2 -15779.118} C_VEL
LIN {X 0,Y 303.473,Z 457.096,A -85,B 0,C 180,E1 -15780.225,E2 -15780.225} C_VEL
LIN {X 0,Y 303.435,Z 456.944,A -85,B 0,C 180,E1 -15780.599,E2 -15780.599} C_VEL
LIN {X 0,Y 303.83,Z 454.773,A -85,B 0,C 180,E1 -15783.619,E2 -15783.619} C_VEL
LIN {X 0,Y 304.447,Z 451.855,A -85,B 0,C 180,E1 -15786.102,E2 -15786.102} C_VEL
LIN {X 0,Y 305.189,Z 448.022,A -85,B 0,C 180,E1 -15788.466,E2 -15788.466} C_VEL
LIN {X 0,Y 306.403,Z 442.381,A -85,B 0,C 180,E1 -15791.15,E2 -15791.15} C_VEL
LIN {X 0,Y 307.924,Z 435.672,A -85,B 0,C 180,E1 -15793.663,E2 -15793.663} C_VEL
LIN {X 0,Y 309.943,Z 427.546,A -85,B 0,C 180,E1 -15796.113,E2 -15796.113} C_VEL
LIN {X 0,Y 312.327,Z 418.081,A -85,B 0,C 180,E1 -15798.434,E2 -15798.434} C_VEL
LIN {X 0,Y 314.637,Z 408.357,A -85,B 0,C 180,E1 -15800.41,E2 -15800.41} C_VEL
LIN {X 0,Y 317.122,Z 397.629,A -85,B 0,C 180,E1 -15802.222,E2 -15802.222} C_VEL
LIN {X 0,Y 319.548,Z 386.228,A -85,B 0,C 180,E1 -15803.827,E2 -15803.827} C_VEL
LIN {X 0,Y 322.059,Z 373.314,A -85,B 0,C 180,E1 -15805.316,E2 -15805.316} C_VEL
LIN {X 0,Y 324.469,Z 358.962,A -85,B 0,C 180,E1 -15806.643,E2 -15806.643} C_VEL
LIN {X 0,Y 326.522,Z 344.475,A -85,B 0,C 180,E1 -15807.685,E2 -15807.685} C_VEL
LIN {X 0,Y 328.124,Z 329.365,A -85,B 0,C 180,E1 -15808.507,E2 -15808.507} C_VEL
LIN {X 0,Y 329.334,Z 314.054,A -85,B 0,C 180,E1 -15809.076,E2 -15809.076} C_VEL
LIN {X 0,Y 331.577,Z 257.307,A -85,B 0,C 180,E1 -15810.395,E2 -15810.395} C_VEL
LIN {X 0,Y 329.139,Z 258.562,A -85,B 0,C 180,E1 -15810.676,E2 -15810.676} C_VEL
LIN {X 0,Y 328.655,Z 258.696,A -85,B 0,C 180,E1 -15810.736,E2 -15810.736} C_VEL
LIN {X 0,Y 325.175,Z 269.146,A -85,B 0,C 180,E1 -15810.902,E2 -15810.902} C_VEL
LIN {X 0,Y 322.645,Z 274.195,A -85,B 0,C 180,E1 -15811.098,E2 -15811.098} C_VEL
LIN {X 0,Y 320.814,Z 276.117,A -85,B 0,C 180,E1 -15811.293,E2 -15811.293} C_VEL
LIN {X 0,Y 319.675,Z 276.272,A -85,B 0,C 180,E1 -15811.447,E2 -15811.447} C_VEL
LIN {X 0,Y 318.789,Z 275.036,A -85,B 0,C 180,E1 -15811.607,E2 -15811.607} C_VEL
LIN {X 0,Y 317.972,Z 272.182,A -85,B 0,C 180,E1 -15811.806,E2 -15811.806} C_VEL
LIN {X 0,Y 317.888,Z 271.332,A -85,B 0,C 180,E1 -15811.843,E2 -15811.843} C_VEL
LIN {X 0,Y 316.578,Z 295.817,A -85,B 0,C 180,E1 -15812.748,E2 -15812.748} C_VEL
LIN {X 0,Y 315.566,Z 312.429,A -85,B 0,C 180,E1 -15813.638,E2 -15813.638} C_VEL
LIN {X 0,Y 314.285,Z 327.213,A -85,B 0,C 180,E1 -15814.68,E2 -15814.68} C_VEL
LIN {X 0,Y 312.905,Z 341.824,A -85,B 0,C 180,E1 -15815.977,E2 -15815.977} C_VEL
LIN {X 0,Y 311.466,Z 355.344,A -85,B 0,C 180,E1 -15817.443,E2 -15817.443} C_VEL
LIN {X 0,Y 310.054,Z 367.923,A -85,B 0,C 180,E1 -15819.083,E2 -15819.083} C_VEL
LIN {X 0,Y 308.516,Z 380.535,A -85,B 0,C 180,E1 -15821.057,E2 -15821.057} C_VEL
LIN {X 0,Y 307.281,Z 391.162,A -85,B 0,C 180,E1 -15823.045,E2 -15823.045} C_VEL
LIN {X 0,Y 306.188,Z 401.542,A -85,B 0,C 180,E1 -15825.375,E2 -15825.375} C_VEL
LIN {X 0,Y 305.229,Z 410.15,A -85,B 0,C 180,E1 -15827.702,E2 -15827.702} C_VEL
LIN {X 0,Y 304.612,Z 417.284,A -85,B 0,C 180,E1 -15830.035,E2 -15830.035} C_VEL
LIN {X 0,Y 304.155,Z 423.813,A -85,B 0,C 180,E1 -15832.698,E2 -15832.698} C_VEL
LIN {X 0,Y 303.941,Z 428.804,A -85,B 0,C 180,E1 -15835.358,E2 -15835.358} C_VEL
LIN {X 0,Y 303.865,Z 431.616,A -85,B 0,C 180,E1 -15837.348,E2 -15837.348} C_VEL
LIN {X 0,Y 303.865,Z 434.223,A -85,B 0,C 180,E1 -15840,E2 -15840} C_VEL
LIN {X 0,Y 304.152,Z 435.571,A -85,B 0,C 180,E1 -15842.648,E2 -15842.648} C_VEL
LIN {X 0,Y 304.397,Z 435.705,A -85,B 0,C 180,E1 -15845.299,E2 -15845.299} C_VEL
LIN {X 0,Y 305.242,Z 434.499,A -85,B 0,C 180,E1 -15848.09,E2 -15848.09} C_VEL
LIN {X 0,Y 306.256,Z 432.304,A -85,B 0,C 180,E1 -15850.578,E2 -15850.578} C_VEL
LIN {X 0,Y 307.544,Z 428.75,A -85,B 0,C 180,E1 -15853.21,E2 -15853.21} C_VEL
LIN {X 0,Y 309.481,Z 423.873,A -85,B 0,C 180,E1 -15855.813,E2 -15855.813} C_VEL
LIN {X 0,Y 311.932,Z 417.602,A -85,B 0,C 180,E1 -15858.386,E2 -15858.386} C_VEL
LIN {X 0,Y 314.952,Z 409.782,A -85,B 0,C 180,E1 -15860.918,E2 -15860.918} C_VEL
LIN {X 0,Y 318.473,Z 400.222,A -85,B 0,C 180,E1 -15863.404,E2 -15863.404} C_VEL
LIN {X 0,Y 322.091,Z 390.127,A -85,B 0,C 180,E1 -15865.527,E2 -15865.527} C_VEL
LIN {X 0,Y 326.114,Z 378.063,A -85,B 0,C 180,E1 -15867.613,E2 -15867.613} C_VEL
LIN {X 0,Y 329.868,Z 365.975,A -85,B 0,C 180,E1 -15869.342,E2 -15869.342} C_VEL
LIN {X 0,Y 334.019,Z 351.563,A -85,B 0,C 180,E1 -15871.03,E2 -15871.03} C_VEL
LIN {X 0,Y 337.332,Z 338.709,A -85,B 0,C 180,E1 -15872.267,E2 -15872.267} C_VEL
LIN {X 0,Y 340.935,Z 323.248,A -85,B 0,C 180,E1 -15873.464,E2 -15873.464} C_VEL
LIN {X 0,Y 344.088,Z 307.16,A -85,B 0,C 180,E1 -15874.438,E2 -15874.438} C_VEL
LIN {X 0,Y 346.718,Z 291.184,A -85,B 0,C 180,E1 -15875.155,E2 -15875.155} C_VEL
LIN {X 0,Y 358.683,Z 221.578,A -85,B 0,C 180,E1 -15877.825,E2 -15877.825} C_VEL
LIN {X 0,Y 361.401,Z 207.065,A -85,B 0,C 180,E1 -15878.382,E2 -15878.382} C_VEL
LIN {X 0,Y 360.055,Z 204.506,A -85,B 0,C 180,E1 -15879.483,E2 -15879.483} C_VEL
LIN {X 0,Y 359.049,Z 202.851,A -85,B 0,C 180,E1 -15880.454,E2 -15880.454} C_VEL
LIN {X 0,Y 357.772,Z 201.005,A -85,B 0,C 180,E1 -15882.211,E2 -15882.211} C_VEL
LIN {X 0,Y 356.939,Z 201.249,A -85,B 0,C 180,E1 -15884.441,E2 -15884.441} C_VEL
LIN {X 0,Y 357.046,Z 202.823,A -85,B 0,C 180,E1 -15886.163,E2 -15886.163} C_VEL
LIN {X 0,Y 357.704,Z 205.303,A -85,B 0,C 180,E1 -15887.716,E2 -15887.716} C_VEL
LIN {X 0,Y 358.887,Z 210.217,A -85,B 0,C 180,E1 -15889.498,E2 -15889.498} C_VEL
LIN {X 0,Y 359.948,Z 214.615,A -85,B 0,C 180,E1 -15890.659,E2 -15890.659} C_VEL
LIN {X 0,Y 359.938,Z 216.256,A -85,B 0,C 180,E1 -15890.864,E2 -15890.864} C_VEL
LIN {X 0,Y 359.601,Z 220.856,A -85,B 0,C 180,E1 -15891.253,E2 -15891.253} C_VEL
LIN {X 0,Y 347.344,Z 293.03,A -85,B 0,C 180,E1 -15893.982,E2 -15893.982} C_VEL
LIN {X 0,Y 342.746,Z 321.984,A -85,B 0,C 180,E1 -15895.14,E2 -15895.14} C_VEL
LIN {X 0,Y 339.037,Z 339.692,A -85,B 0,C 180,E1 -15896.055,E2 -15896.055} C_VEL
LIN {X 0,Y 335.029,Z 355.777,A -85,B 0,C 180,E1 -15897.126,E2 -15897.126} C_VEL
LIN {X 0,Y 330.928,Z 370.791,A -85,B 0,C 180,E1 -15898.397,E2 -15898.397} C_VEL
LIN {X 0,Y 326.566,Z 385.746,A -85,B 0,C 180,E1 -15899.976,E2 -15899.976} C_VEL
LIN {X 0,Y 322.089,Z 400.165,A -85,B 0,C 180,E1 -15901.845,E2 -15901.845} C_VEL
LIN {X 0,Y 318.322,Z 412.353,A -85,B 0,C 180,E1 -15903.796,E2 -15903.796} C_VEL
LIN {X 0,Y 314.652,Z 423.612,A -85,B 0,C 180,E1 -15905.944,E2 -15905.944} C_VEL
LIN {X 0,Y 311.704,Z 433.171,A -85,B 0,C 180,E1 -15908.159,E2 -15908.159} C_VEL
LIN {X 0,Y 308.867,Z 442.416,A -85,B 0,C 180,E1 -15910.735,E2 -15910.735} C_VEL
LIN {X 0,Y 305.899,Z 454.446,A -85,B 0,C 180,E1 -15914.783,E2 -15914.783} C_VEL
LIN {X 0,Y 304.822,Z 460.69,A -85,B 0,C 180,E1 -15917.348,E2 -15917.348} C_VEL
LIN {X 0,Y 304.067,Z 465.751,A -85,B 0,C 180,E1 -15920.017,E2 -15920.017} C_VEL
LIN {X 0,Y 303.791,Z 468.69,A -85,B 0,C 180,E1 -15922.021,E2 -15922.021} C_VEL
LIN {X 0,Y 303.615,Z 471.461,A -85,B 0,C 180,E1 -15924.687,E2 -15924.687} C_VEL
LIN {X 0,Y 303.631,Z 473.024,A -85,B 0,C 180,E1 -15927.347,E2 -15927.347} C_VEL
LIN {X 0,Y 303.607,Z 473.395,A -85,B 0,C 180,E1 -15930,E2 -15930} C_VEL
LIN {X 0,Y 303.633,Z 472.577,A -85,B 0,C 180,E1 -15932.653,E2 -15932.653} C_VEL
LIN {X 0,Y 303.615,Z 470.543,A -85,B 0,C 180,E1 -15935.313,E2 -15935.313} C_VEL
LIN {X 0,Y 303.798,Z 467.24,A -85,B 0,C 180,E1 -15937.979,E2 -15937.979} C_VEL
LIN {X 0,Y 304.091,Z 462.576,A -85,B 0,C 180,E1 -15940.655,E2 -15940.655} C_VEL
LIN {X 0,Y 304.89,Z 456.464,A -85,B 0,C 180,E1 -15943.327,E2 -15943.327} C_VEL
LIN {X 0,Y 307.097,Z 446.597,A -85,B 0,C 180,E1 -15947.308,E2 -15947.308} C_VEL
LIN {X 0,Y 309.395,Z 438.5,A -85,B 0,C 180,E1 -15949.921,E2 -15949.921} C_VEL
LIN {X 0,Y 312.256,Z 428.757,A -85,B 0,C 180,E1 -15952.496,E2 -15952.496} C_VEL
LIN {X 0,Y 315.445,Z 418.594,A -85,B 0,C 180,E1 -15954.692,E2 -15954.692} C_VEL
LIN {X 0,Y 319.266,Z 406.587,A -85,B 0,C 180,E1 -15956.825,E2 -15956.825} C_VEL
LIN {X 0,Y 322.97,Z 394.635,A -85,B 0,C 180,E1 -15958.603,E2 -15958.603} C_VEL
LIN {X 0,Y 327.251,Z 380.508,A -85,B 0,C 180,E1 -15960.31,E2 -15960.31} C_VEL
LIN {X 0,Y 331.186,Z 366.317,A -85,B 0,C 180,E1 -15961.725,E2 -15961.725} C_VEL
LIN {X 0,Y 335.048,Z 351.892,A -85,B 0,C 180,E1 -15962.872,E2 -15962.872} C_VEL
LIN {X 0,Y 338.778,Z 335.884,A -85,B 0,C 180,E1 -15963.885,E2 -15963.885} C_VEL
LIN {X 0,Y 342.428,Z 317.773,A -85,B 0,C 180,E1 -15964.763,E2 -15964.763} C_VEL
LIN {X 0,Y 355.596,Z 235.971,A -85,B 0,C 180,E1 -15967.911,E2 -15967.911} C_VEL
LIN {X 0,Y 359.473,Z 214.089,A -85,B 0,C 180,E1 -15968.758,E2 -15968.758} C_VEL
LIN {X 0,Y 360.617,Z 203.974,A -85,B 0,C 180,E1 -15969.478,E2 -15969.478} C_VEL
LIN {X 0,Y 360.477,Z 202.1,A -85,B 0,C 180,E1 -15969.798,E2 -15969.798} C_VEL
LIN {X 0,Y 359.089,Z 198.993,A -85,B 0,C 180,E1 -15971.118,E2 -15971.118} C_VEL
LIN {X 0,Y 357.951,Z 196.246,A -85,B 0,C 180,E1 -15972.699,E2 -15972.699} C_VEL
LIN {X 0,Y 357.063,Z 194.91,A -85,B 0,C 180,E1 -15974.881,E2 -15974.881} C_VEL
LIN {X 0,Y 357.306,Z 195.075,A -85,B 0,C 180,E1 -15977.036,E2 -15977.036} C_VEL
LIN {X 0,Y 358.332,Z 196.644,A -85,B 0,C 180,E1 -15978.847,E2 -15978.847} C_VEL
LIN {X 0,Y 359.722,Z 199.767,A -85,B 0,C 180,E1 -15980.482,E2 -15980.482} C_VEL
LIN {X 0,Y 361.088,Z 203.031,A -85,B 0,C 180,E1 -15981.676,E2 -15981.676} C_VEL
LIN {X 0,Y 348.765,Z 273.578,A -85,B 0,C 180,E1 -15984.374,E2 -15984.374} C_VEL
LIN {X 0,Y 344.904,Z 298.411,A -85,B 0,C 180,E1 -15985.345,E2 -15985.345} C_VEL
LIN {X 0,Y 341.96,Z 314.965,A -85,B 0,C 180,E1 -15986.208,E2 -15986.208} C_VEL
LIN {X 0,Y 338.923,Z 329.531,A -85,B 0,C 180,E1 -15987.199,E2 -15987.199} C_VEL
LIN {X 0,Y 335.065,Z 345.305,A -85,B 0,C 180,E1 -15988.55,E2 -15988.55} C_VEL
LIN {X 0,Y 331.241,Z 359.543,A -85,B 0,C 180,E1 -15990.093,E2 -15990.093} C_VEL
LIN {X 0,Y 327.33,Z 372.651,A -85,B 0,C 180,E1 -15991.813,E2 -15991.813} C_VEL
LIN {X 0,Y 323.728,Z 383.793,A -85,B 0,C 180,E1 -15993.574,E2 -15993.574} C_VEL
LIN {X 0,Y 320.418,Z 393.377,A -85,B 0,C 180,E1 -15995.371,E2 -15995.371} C_VEL
LIN {X 0,Y 317.055,Z 402.873,A -85,B 0,C 180,E1 -15997.52,E2 -15997.52} C_VEL
LIN {X 0,Y 313.837,Z 411.867,A -85,B 0,C 180,E1 -16000.032,E2 -16000.032} C_VEL
LIN {X 0,Y 311.295,Z 418.391,A -85,B 0,C 180,E1 -16002.255,E2 -16002.255} C_VEL
LIN {X 0,Y 309.448,Z 423.092,A -85,B 0,C 180,E1 -16004.185,E2 -16004.185} C_VEL
LIN {X 0,Y 307.553,Z 428.041,A -85,B 0,C 180,E1 -16006.791,E2 -16006.791} C_VEL
LIN {X 0,Y 306.249,Z 431.643,A -85,B 0,C 180,E1 -16009.422,E2 -16009.422} C_VEL
LIN {X 0,Y 305.06,Z 434.102,A -85,B 0,C 180,E1 -16012.155,E2 -16012.155} C_VEL
LIN {X 0,Y 304.36,Z 435.192,A -85,B 0,C 180,E1 -16014.701,E2 -16014.701} C_VEL
LIN {X 0,Y 304.117,Z 435.122,A -85,B 0,C 180,E1 -16017.351,E2 -16017.351} C_VEL
LIN {X 0,Y 303.855,Z 433.831,A -85,B 0,C 180,E1 -16020,E2 -16020} C_VEL
LIN {X 0,Y 303.828,Z 431.275,A -85,B 0,C 180,E1 -16022.652,E2 -16022.652} C_VEL
LIN {X 0,Y 303.947,Z 427.385,A -85,B 0,C 180,E1 -16025.307,E2 -16025.307} C_VEL
LIN {X 0,Y 304.285,Z 422.069,A -85,B 0,C 180,E1 -16027.966,E2 -16027.966} C_VEL
LIN {X 0,Y 304.721,Z 415.167,A -85,B 0,C 180,E1 -16030.633,E2 -16030.633} C_VEL
LIN {X 0,Y 305.473,Z 407.686,A -85,B 0,C 180,E1 -16032.963,E2 -16032.963} C_VEL
LIN {X 0,Y 306.251,Z 398.642,A -85,B 0,C 180,E1 -16035.294,E2 -16035.294} C_VEL
LIN {X 0,Y 307.561,Z 387.692,A -85,B 0,C 180,E1 -16037.625,E2 -16037.625} C_VEL
LIN {X 0,Y 308.915,Z 376.495,A -85,B 0,C 180,E1 -16039.608,E2 -16039.608} C_VEL
LIN {X 0,Y 310.314,Z 364.16,A -85,B 0,C 180,E1 -16041.44,E2 -16041.44} C_VEL
LIN {X 0,Y 311.864,Z 351.12,A -85,B 0,C 180,E1 -16043.052,E2 -16043.052} C_VEL
LIN {X 0,Y 313.312,Z 336.777,A -85,B 0,C 180,E1 -16044.519,E2 -16044.519} C_VEL
LIN {X 0,Y 314.676,Z 322.088,A -85,B 0,C 180,E1 -16045.73,E2 -16045.73} C_VEL
LIN {X 0,Y 315.887,Z 305.756,A -85,B 0,C 180,E1 -16046.778,E2 -16046.778} C_VEL
LIN {X 0,Y 316.833,Z 289.342,A -85,B 0,C 180,E1 -16047.551,E2 -16047.551} C_VEL
LIN {X 0,Y 322.59,Z 173.498,A -85,B 0,C 180,E1 -16051.243,E2 -16051.243} C_VEL
LIN {X 0,Y 305.629,Z 133.876,A -85,B 0,C 180,E1 -16053.954,E2 -16053.954} C_VEL
LIN {X 0,Y 305.484,Z 133.058,A -85,B 0,C 180,E1 -16054.027,E2 -16054.027} C_VEL
LIN {X 0,Y 305.456,Z 133.06,A -85,B 0,C 180,E1 -16056.743,E2 -16056.743} C_VEL
LIN {X 0,Y 305.411,Z 133.066,A -85,B 0,C 180,E1 -16060.59,E2 -16060.59} C_VEL
LIN {X 0,Y 305.422,Z 133.059,A -85,B 0,C 180,E1 -16063.656,E2 -16063.656} C_VEL
LIN {X 0,Y 305.436,Z 133.032,A -85,B 0,C 180,E1 -16067.419,E2 -16067.419} C_VEL
LIN {X 0,Y 305.462,Z 133.057,A -85,B 0,C 180,E1 -16071.595,E2 -16071.595} C_VEL
LIN {X 0,Y 305.463,Z 133.035,A -85,B 0,C 180,E1 -16074.887,E2 -16074.887} C_VEL
LIN {X 0,Y 305.444,Z 133.063,A -85,B 0,C 180,E1 -16078.358,E2 -16078.358} C_VEL
LIN {X 0,Y 305.478,Z 133.04,A -85,B 0,C 180,E1 -16081.109,E2 -16081.109} C_VEL
LIN {X 0,Y 305.483,Z 133.058,A -85,B 0,C 180,E1 -16084.08,E2 -16084.08} C_VEL
LIN {X 0,Y 305.463,Z 133.062,A -85,B 0,C 180,E1 -16088.4,E2 -16088.4} C_VEL
LIN {X 0,Y 305.512,Z 133.048,A -85,B 0,C 180,E1 -16091.213,E2 -16091.213} C_VEL
LIN {X 0,Y 305.582,Z 133.048,A -85,B 0,C 180,E1 -16095.346,E2 -16095.346} C_VEL
LIN {X 0,Y 305.611,Z 133.158,A -85,B 0,C 180,E1 -16097.128,E2 -16097.128} C_VEL
LIN {X 0,Y 309.726,Z 145.348,A -85,B 0,C 180,E1 -16100.013,E2 -16100.013} C_VEL
LIN {X 0,Y 317.663,Z 160.937,A -85,B 0,C 180,E1 -16101.404,E2 -16101.404} C_VEL
LIN {X 0,Y 326.644,Z 180.859,A -85,B 0,C 180,E1 -16102.945,E2 -16102.945} C_VEL
LIN {X 0,Y 329.381,Z 188.063,A -85,B 0,C 180,E1 -16103.423,E2 -16103.423} C_VEL
LIN {X 0,Y 325.113,Z 311.914,A -85,B 0,C 180,E1 -16106.204,E2 -16106.204} C_VEL
LIN {X 0,Y 324.054,Z 327.189,A -85,B 0,C 180,E1 -16106.754,E2 -16106.754} C_VEL
LIN {X 0,Y 322.672,Z 342.632,A -85,B 0,C 180,E1 -16107.581,E2 -16107.581} C_VEL
LIN {X 0,Y 320.978,Z 356.829,A -85,B 0,C 180,E1 -16108.589,E2 -16108.589} C_VEL
LIN {X 0,Y 319.018,Z 370.676,A -85,B 0,C 180,E1 -16109.842,E2 -16109.842} C_VEL
LIN {X 0,Y 316.888,Z 383.451,A -85,B 0,C 180,E1 -16111.271,E2 -16111.271} C_VEL
LIN {X 0,Y 314.561,Z 396.326,A -85,B 0,C 180,E1 -16113.042,E2 -16113.042} C_VEL
LIN {X 0,Y 312.457,Z 407.129,A -85,B 0,C 180,E1 -16114.839,E2 -16114.839} C_VEL
LIN {X 0,Y 310.465,Z 417.091,A -85,B 0,C 180,E1 -16116.825,E2 -16116.825} C_VEL
LIN {X 0,Y 308.437,Z 426.826,A -85,B 0,C 180,E1 -16119.178,E2 -16119.178} C_VEL
LIN {X 0,Y 306.885,Z 434.778,A -85,B 0,C 180,E1 -16121.526,E2 -16121.526} C_VEL
LIN {X 0,Y 305.648,Z 441.527,A -85,B 0,C 180,E1 -16123.971,E2 -16123.971} C_VEL
LIN {X 0,Y 304.613,Z 447.584,A -85,B 0,C 180,E1 -16126.762,E2 -16126.762} C_VEL
LIN {X 0,Y 304.08,Z 451.171,A -85,B 0,C 180,E1 -16128.879,E2 -16128.879} C_VEL
LIN {X 0,Y 303.557,Z 454.713,A -85,B 0,C 180,E1 -16131.742,E2 -16131.742} C_VEL
LIN {X 0,Y 303.336,Z 456.866,A -85,B 0,C 180,E1 -16134.648,E2 -16134.648} C_VEL
LIN {X 0,Y 303.29,Z 457.632,A -85,B 0,C 180,E1 -16137.61,E2 -16137.61} C_VEL
LIN {X 0,Y 303.348,Z 457.472,A -85,B 0,C 180,E1 -16139.113,E2 -16139.113} C_VEL
LIN {X 0,Y 303.435,Z 456.944,A -85,B 0,C 180,E1 -16140.599,E2 -16140.599} C_VEL
LIN {X 0,Y 302.917,Z 456.437,A -85,B 0,C 180,E1 -16141.705,E2 -16141.705} C_VEL
LIN {X 0,Y 300.339,Z 455.155,A -85,B 0,C 180,E1 -16143.507,E2 -16143.507} C_VEL
LIN {X 0,Y 298.208,Z 453.743,A -85,B 0,C 180,E1 -16144.957,E2 -16144.957} C_VEL
LIN {X 0,Y 297.445,Z 452.439,A -85,B 0,C 180,E1 -16146.064,E2 -16146.064} C_VEL
LIN {X 0,Y 297.466,Z 451.962,A -85,B 0,C 180,E1 -16146.435,E2 -16146.435} C_VEL
LIN {X 0,Y 298.32,Z 447.902,A -85,B 0,C 180,E1 -16148.973,E2 -16148.973} C_VEL
LIN {X 0,Y 299.796,Z 441.583,A -85,B 0,C 180,E1 -16151.97,E2 -16151.97} C_VEL
LIN {X 0,Y 301.663,Z 433.958,A -85,B 0,C 180,E1 -16154.755,E2 -16154.755} C_VEL
LIN {X 0,Y 303.937,Z 425.449,A -85,B 0,C 180,E1 -16157.236,E2 -16157.236} C_VEL
LIN {X 0,Y 306.478,Z 415.57,A -85,B 0,C 180,E1 -16159.585,E2 -16159.585} C_VEL
LIN {X 0,Y 309.077,Z 404.882,A -85,B 0,C 180,E1 -16161.673,E2 -16161.673} C_VEL
LIN {X 0,Y 311.731,Z 393.924,A -85,B 0,C 180,E1 -16163.434,E2 -16163.434} C_VEL
LIN {X 0,Y 314.351,Z 381.896,A -85,B 0,C 180,E1 -16165.035,E2 -16165.035} C_VEL
LIN {X 0,Y 316.875,Z 368.745,A -85,B 0,C 180,E1 -16166.464,E2 -16166.464} C_VEL
LIN {X 0,Y 319.285,Z 354.023,A -85,B 0,C 180,E1 -16167.735,E2 -16167.735} C_VEL
LIN {X 0,Y 321.24,Z 339.286,A -85,B 0,C 180,E1 -16168.716,E2 -16168.716} C_VEL
LIN {X 0,Y 322.731,Z 324.78,A -85,B 0,C 180,E1 -16169.426,E2 -16169.426} C_VEL
LIN {X 0,Y 323.821,Z 309.399,A -85,B 0,C 180,E1 -16169.932,E2 -16169.932} C_VEL
LIN {X 0,Y 324.848,Z 280.835,A -85,B 0,C 180,E1 -16170.615,E2 -16170.615} C_VEL
LIN {X 0,Y 322.072,Z 282.814,A -85,B 0,C 180,E1 -16170.929,E2 -16170.929} C_VEL
LIN {X 0,Y 320.669,Z 283.309,A -85,B 0,C 180,E1 -16171.105,E2 -16171.105} C_VEL
LIN {X 0,Y 317.341,Z 292.568,A -85,B 0,C 180,E1 -16171.294,E2 -16171.294} C_VEL
LIN {X 0,Y 314.466,Z 297.457,A -85,B 0,C 180,E1 -16171.555,E2 -16171.555} C_VEL
LIN {X 0,Y 312.793,Z 298.897,A -85,B 0,C 180,E1 -16171.754,E2 -16171.754} C_VEL
LIN {X 0,Y 311.379,Z 298.881,A -85,B 0,C 180,E1 -16171.962,E2 -16171.962} C_VEL
LIN {X 0,Y 310.446,Z 297.611,A -85,B 0,C 180,E1 -16172.14,E2 -16172.14} C_VEL
LIN {X 0,Y 309.84,Z 294.312,A -85,B 0,C 180,E1 -16172.335,E2 -16172.335} C_VEL
LIN {X 0,Y 308.818,Z 310.616,A -85,B 0,C 180,E1 -16173.199,E2 -16173.199} C_VEL
LIN {X 0,Y 307.417,Z 326.908,A -85,B 0,C 180,E1 -16174.345,E2 -16174.345} C_VEL
LIN {X 0,Y 305.911,Z 342.44,A -85,B 0,C 180,E1 -16175.753,E2 -16175.753} C_VEL
LIN {X 0,Y 304.314,Z 357.036,A -85,B 0,C 180,E1 -16177.395,E2 -16177.395} C_VEL
LIN {X 0,Y 302.787,Z 370.695,A -85,B 0,C 180,E1 -16179.269,E2 -16179.269} C_VEL
LIN {X 0,Y 301.25,Z 382.934,A -85,B 0,C 180,E1 -16181.289,E2 -16181.289} C_VEL
LIN {X 0,Y 300.017,Z 393.263,A -85,B 0,C 180,E1 -16183.323,E2 -16183.323} C_VEL
LIN {X 0,Y 298.904,Z 403.382,A -85,B 0,C 180,E1 -16185.706,E2 -16185.706} C_VEL
LIN {X 0,Y 298.093,Z 410.655,A -85,B 0,C 180,E1 -16187.749,E2 -16187.749} C_VEL
LIN {X 0,Y 297.554,Z 416.866,A -85,B 0,C 180,E1 -16189.796,E2 -16189.796} C_VEL
LIN {X 0,Y 297.088,Z 423.6,A -85,B 0,C 180,E1 -16192.524,E2 -16192.524} C_VEL
LIN {X 0,Y 296.863,Z 428.775,A -85,B 0,C 180,E1 -16195.247,E2 -16195.247} C_VEL
LIN {X 0,Y 296.784,Z 431.682,A -85,B 0,C 180,E1 -16197.285,E2 -16197.285} C_VEL
LIN {X 0,Y 296.769,Z 434.458,A -85,B 0,C 180,E1 -16200,E2 -16200} C_VEL
LIN {X 0,Y 297.065,Z 435.975,A -85,B 0,C 180,E1 -16202.712,E2 -16202.712} C_VEL
LIN {X 0,Y 297.352,Z 436.286,A -85,B 0,C 180,E1 -16205.424,E2 -16205.424} C_VEL
LIN {X 0,Y 298.223,Z 435.31,A -85,B 0,C 180,E1 -16208.197,E2 -16208.197} C_VEL
LIN {X 0,Y 299.321,Z 433.184,A -85,B 0,C 180,E1 -16210.826,E2 -16210.826} C_VEL
LIN {X 0,Y 300.712,Z 429.827,A -85,B 0,C 180,E1 -16213.515,E2 -16213.515} C_VEL
LIN {X 0,Y 302.766,Z 425.173,A -85,B 0,C 180,E1 -16216.173,E2 -16216.173} C_VEL
LIN {X 0,Y 305.365,Z 419.152,A -85,B 0,C 180,E1 -16218.796,E2 -16218.796} C_VEL
LIN {X 0,Y 308.574,Z 411.613,A -85,B 0,C 180,E1 -16221.371,E2 -16221.371} C_VEL
LIN {X 0,Y 312.267,Z 402.415,A -85,B 0,C 180,E1 -16223.898,E2 -16223.898} C_VEL
LIN {X 0,Y 316.069,Z 392.723,A -85,B 0,C 180,E1 -16226.05,E2 -16226.05} C_VEL
LIN {X 0,Y 320.329,Z 381.201,A -85,B 0,C 180,E1 -16228.155,E2 -16228.155} C_VEL
LIN {X 0,Y 324.57,Z 368.681,A -85,B 0,C 180,E1 -16230.048,E2 -16230.048} C_VEL
LIN {X 0,Y 328.948,Z 354.818,A -85,B 0,C 180,E1 -16231.743,E2 -16231.743} C_VEL
LIN {X 0,Y 332.835,Z 341.138,A -85,B 0,C 180,E1 -16233.118,E2 -16233.118} C_VEL
LIN {X 0,Y 336.609,Z 326.331,A -85,B 0,C 180,E1 -16234.314,E2 -16234.314} C_VEL
LIN {X 0,Y 340.173,Z 310.142,A -85,B 0,C 180,E1 -16235.344,E2 -16235.344} C_VEL
LIN {X 0,Y 343.135,Z 293.795,A -85,B 0,C 180,E1 -16236.12,E2 -16236.12} C_VEL
LIN {X 0,Y 356.251,Z 222.673,A -85,B 0,C 180,E1 -16238.879,E2 -16238.879} C_VEL
LIN {X 0,Y 358.409,Z 212.008,A -85,B 0,C 180,E1 -16239.281,E2 -16239.281} C_VEL
LIN {X 0,Y 357.044,Z 209.55,A -85,B 0,C 180,E1 -16240.651,E2 -16240.651} C_VEL
LIN {X 0,Y 356.014,Z 207.869,A -85,B 0,C 180,E1 -16242.158,E2 -16242.158} C_VEL
LIN {X 0,Y 355.14,Z 208.135,A -85,B 0,C 180,E1 -16244.445,E2 -16244.445} C_VEL
LIN {X 0,Y 355.192,Z 209.746,A -85,B 0,C 180,E1 -16246.096,E2 -16246.096} C_VEL
LIN {X 0,Y 355.66,Z 211.89,A -85,B 0,C 180,E1 -16247.429,E2 -16247.429} C_VEL
LIN {X 0,Y 356.572,Z 216.402,A -85,B 0,C 180,E1 -16249.074,E2 -16249.074} C_VEL
LIN {X 0,Y 357.223,Z 219.724,A -85,B 0,C 180,E1 -16249.974,E2 -16249.974} C_VEL
LIN {X 0,Y 356.845,Z 223.081,A -85,B 0,C 180,E1 -16250.249,E2 -16250.249} C_VEL
LIN {X 0,Y 344.056,Z 293.488,A -85,B 0,C 180,E1 -16252.944,E2 -16252.944} C_VEL
LIN {X 0,Y 339.241,Z 321.361,A -85,B 0,C 180,E1 -16254.079,E2 -16254.079} C_VEL
LIN {X 0,Y 335.565,Z 337.818,A -85,B 0,C 180,E1 -16254.925,E2 -16254.925} C_VEL
LIN {X 0,Y 331.33,Z 353.903,A -85,B 0,C 180,E1 -16255.982,E2 -16255.982} C_VEL
LIN {X 0,Y 326.759,Z 369.492,A -85,B 0,C 180,E1 -16257.29,E2 -16257.29} C_VEL
LIN {X 0,Y 322.276,Z 383.865,A -85,B 0,C 180,E1 -16258.807,E2 -16258.807} C_VEL
LIN {X 0,Y 317.816,Z 397.265,A -85,B 0,C 180,E1 -16260.526,E2 -16260.526} C_VEL
LIN {X 0,Y 313.874,Z 408.804,A -85,B 0,C 180,E1 -16262.315,E2 -16262.315} C_VEL
LIN {X 0,Y 309.805,Z 420.399,A -85,B 0,C 180,E1 -16264.468,E2 -16264.468} C_VEL
LIN {X 0,Y 305.974,Z 431.588,A -85,B 0,C 180,E1 -16267.016,E2 -16267.016} C_VEL
LIN {X 0,Y 302.866,Z 440.938,A -85,B 0,C 180,E1 -16269.63,E2 -16269.63} C_VEL
LIN {X 0,Y 300.385,Z 448.674,A -85,B 0,C 180,E1 -16272.293,E2 -16272.293} C_VEL
LIN {X 0,Y 298.381,Z 457.578,A -85,B 0,C 180,E1 -16275.681,E2 -16275.681} C_VEL
LIN {X 0,Y 297.349,Z 463.317,A -85,B 0,C 180,E1 -16278.41,E2 -16278.41} C_VEL
LIN {X 0,Y 296.901,Z 466.74,A -85,B 0,C 180,E1 -16280.462,E2 -16280.462} C_VEL
LIN {X 0,Y 296.628,Z 470.103,A -85,B 0,C 180,E1 -16283.196,E2 -16283.196} C_VEL
LIN {X 0,Y 296.504,Z 472.236,A -85,B 0,C 180,E1 -16285.922,E2 -16285.922} C_VEL
LIN {X 0,Y 296.509,Z 473.177,A -85,B 0,C 180,E1 -16288.642,E2 -16288.642} C_VEL
LIN {X 0,Y 296.509,Z 472.93,A -85,B 0,C 180,E1 -16291.358,E2 -16291.358} C_VEL
LIN {X 0,Y 296.525,Z 471.483,A -85,B 0,C 180,E1 -16294.077,E2 -16294.077} C_VEL
LIN {X 0,Y 296.63,Z 468.798,A -85,B 0,C 180,E1 -16296.803,E2 -16296.803} C_VEL
LIN {X 0,Y 296.839,Z 464.8,A -85,B 0,C 180,E1 -16299.54,E2 -16299.54} C_VEL
LIN {X 0,Y 297.472,Z 459.403,A -85,B 0,C 180,E1 -16302.277,E2 -16302.277} C_VEL
LIN {X 0,Y 298.21,Z 454.768,A -85,B 0,C 180,E1 -16304.327,E2 -16304.327} C_VEL
LIN {X 0,Y 299.782,Z 448.786,A -85,B 0,C 180,E1 -16307.04,E2 -16307.04} C_VEL
LIN {X 0,Y 302.073,Z 441.361,A -85,B 0,C 180,E1 -16309.716,E2 -16309.716} C_VEL
LIN {X 0,Y 304.913,Z 432.412,A -85,B 0,C 180,E1 -16312.33,E2 -16312.33} C_VEL
LIN {X 0,Y 308.081,Z 422.975,A -85,B 0,C 180,E1 -16314.603,E2 -16314.603} C_VEL
LIN {X 0,Y 311.934,Z 411.987,A -85,B 0,C 180,E1 -16316.783,E2 -16316.783} C_VEL
LIN {X 0,Y 316.331,Z 399.015,A -85,B 0,C 180,E1 -16318.896,E2 -16318.896} C_VEL
LIN {X 0,Y 320.64,Z 385.983,A -85,B 0,C 180,E1 -16320.638,E2 -16320.638} C_VEL
LIN {X 0,Y 325.325,Z 370.977,A -85,B 0,C 180,E1 -16322.275,E2 -16322.275} C_VEL
LIN {X 0,Y 329.414,Z 356.875,A -85,B 0,C 180,E1 -16323.507,E2 -16323.507} C_VEL
LIN {X 0,Y 333.798,Z 340.475,A -85,B 0,C 180,E1 -16324.644,E2 -16324.644} C_VEL
LIN {X 0,Y 337.663,Z 323.523,A -85,B 0,C 180,E1 -16325.543,E2 -16325.543} C_VEL
LIN {X 0,Y 341.417,Z 302.294,A -85,B 0,C 180,E1 -16326.423,E2 -16326.423} C_VEL
LIN {X 0,Y 353.787,Z 232.032,A -85,B 0,C 180,E1 -16329.149,E2 -16329.149} C_VEL
LIN {X 0,Y 356.899,Z 215.55,A -85,B 0,C 180,E1 -16329.803,E2 -16329.803} C_VEL
LIN {X 0,Y 357.922,Z 207.962,A -85,B 0,C 180,E1 -16330.36,E2 -16330.36} C_VEL
LIN {X 0,Y 356.848,Z 205.282,A -85,B 0,C 180,E1 -16331.549,E2 -16331.549} C_VEL
LIN {X 0,Y 356.014,Z 202.979,A -85,B 0,C 180,E1 -16332.882,E2 -16332.882} C_VEL
LIN {X 0,Y 355.295,Z 201.882,A -85,B 0,C 180,E1 -16334.594,E2 -16334.594} C_VEL
LIN {X 0,Y 355.371,Z 201.799,A -85,B 0,C 180,E1 -16336.611,E2 -16336.611} C_VEL
LIN {X 0,Y 356.314,Z 203.181,A -85,B 0,C 180,E1 -16338.549,E2 -16338.549} C_VEL
LIN {X 0,Y 357.611,Z 206.443,A -85,B 0,C 180,E1 -16340.256,E2 -16340.256} C_VEL
LIN {X 0,Y 358.133,Z 207.721,A -85,B 0,C 180,E1 -16340.77,E2 -16340.77} C_VEL
LIN {X 0,Y 344.991,Z 278.142,A -85,B 0,C 180,E1 -16343.471,E2 -16343.471} C_VEL
LIN {X 0,Y 341.087,Z 301.117,A -85,B 0,C 180,E1 -16344.403,E2 -16344.403} C_VEL
LIN {X 0,Y 338.144,Z 316.409,A -85,B 0,C 180,E1 -16345.232,E2 -16345.232} C_VEL
LIN {X 0,Y 334.481,Z 332.248,A -85,B 0,C 180,E1 -16346.346,E2 -16346.346} C_VEL
LIN {X 0,Y 330.433,Z 347.45,A -85,B 0,C 180,E1 -16347.698,E2 -16347.698} C_VEL
LIN {X 0,Y 326.033,Z 362.397,A -85,B 0,C 180,E1 -16349.386,E2 -16349.386} C_VEL
LIN {X 0,Y 322.24,Z 374.041,A -85,B 0,C 180,E1 -16350.97,E2 -16350.97} C_VEL
LIN {X 0,Y 317.802,Z 386.666,A -85,B 0,C 180,E1 -16353.042,E2 -16353.042} C_VEL
LIN {X 0,Y 313.826,Z 397.23,A -85,B 0,C 180,E1 -16355.172,E2 -16355.172} C_VEL
LIN {X 0,Y 310.346,Z 406.148,A -85,B 0,C 180,E1 -16357.358,E2 -16357.358} C_VEL
LIN {X 0,Y 306.97,Z 414.59,A -85,B 0,C 180,E1 -16359.915,E2 -16359.915} C_VEL
LIN {X 0,Y 303.958,Z 421.49,A -85,B 0,C 180,E1 -16362.508,E2 -16362.508} C_VEL
LIN {X 0,Y 301.77,Z 426.889,A -85,B 0,C 180,E1 -16365.157,E2 -16365.157} C_VEL
LIN {X 0,Y 300.003,Z 430.975,A -85,B 0,C 180,E1 -16367.829,E2 -16367.829} C_VEL
LIN {X 0,Y 298.681,Z 433.812,A -85,B 0,C 180,E1 -16370.52,E2 -16370.52} C_VEL
LIN {X 0,Y 297.663,Z 435.42,A -85,B 0,C 180,E1 -16373.221,E2 -16373.221} C_VEL
LIN {X 0,Y 297.15,Z 435.787,A -85,B 0,C 180,E1 -16375.932,E2 -16375.932} C_VEL
LIN {X 0,Y 296.84,Z 434.94,A -85,B 0,C 180,E1 -16378.644,E2 -16378.644} C_VEL
LIN {X 0,Y 296.706,Z 432.852,A -85,B 0,C 180,E1 -16381.358,E2 -16381.358} C_VEL
LIN {X 0,Y 296.812,Z 429.469,A -85,B 0,C 180,E1 -16384.074,E2 -16384.074} C_VEL
LIN {X 0,Y 297.025,Z 424.702,A -85,B 0,C 180,E1 -16386.795,E2 -16386.795} C_VEL
LIN {X 0,Y 297.39,Z 418.423,A -85,B 0,C 180,E1 -16389.522,E2 -16389.522} C_VEL
LIN {X 0,Y 297.951,Z 411.543,A -85,B 0,C 180,E1 -16391.912,E2 -16391.912} C_VEL
